EventTableTriggerLogic 9452: layoutX=184, layoutY=128, Operand1=AND 6402, Operand2=AND 6408, Operator=0, Delay=1000
EventTableTriggerLogic 9453: layoutX=184, layoutY=128, Operand1=AND 6402, Operand2=AND 6408, Operator=0, Delay=1000
EventTableTriggerLogic 9454: layoutX=184, layoutY=128, Operand1=AND 6402, Operand2=AND 6408, Operator=0, Delay=1000
EventTableTriggerLogic 9455: layoutX=231, layoutY=144, Operand1=AND 6416, Operand2=pallet1 6426, Operator=0, Delay=1000
EventTableTriggerLogic 9456: layoutX=231, layoutY=144, Operand1=AND 6416, Operand2=pallet1 6426, Operator=0, Delay=1000
EventTableTriggerLogic 9457: layoutX=231, layoutY=144, Operand1=AND 6416, Operand2=pallet1 6426, Operator=0, Delay=1000
EventTableTriggerLogic 9458: layoutX=231, layoutY=144, Operand1=AND 6416, Operand2=pallet1 6426, Operator=0, Delay=1000
EventTableTriggerLogic 9459: layoutX=231, layoutY=144, Operand1=AND 6416, Operand2=pallet1 6426, Operator=0, Delay=1000
EventTableTriggerLogic 9460: layoutX=231, layoutY=144, Operand1=AND 6416, Operand2=pallet1 6426, Operator=0, Delay=1000
EventTableTriggerLogic 9461: layoutX=251, layoutY=143, Operand1=AND 8115, Operand2=pallet3.1 8114, Operator=0, Delay=1000
EventTableTriggerLogic 9462: layoutX=251, layoutY=143, Operand1=AND 8115, Operand2=pallet3.1 8114, Operator=0, Delay=1000
EventTableTriggerLogic 9463: layoutX=251, layoutY=143, Operand1=AND 8115, Operand2=pallet3.1 8114, Operator=0, Delay=1000
EventTableTriggerLogic 9464: layoutX=251, layoutY=143, Operand1=AND 8115, Operand2=pallet3.1 8114, Operator=0, Delay=1000
EventTableTriggerLogic 9465: layoutX=251, layoutY=143, Operand1=AND 8115, Operand2=pallet3.1 8114, Operator=0, Delay=1000
EventTableTriggerLogic 9466: layoutX=251, layoutY=143, Operand1=AND 8115, Operand2=pallet3.1 8114, Operator=0, Delay=1000
EventTableTriggerLogic 9467: layoutX=62, layoutY=38, Operand1=pallet2 8126, Operand2=cellC_slider_horizontal_move 8125, Operator=0, Delay=1000
EventTableTriggerLogic 9468: layoutX=62, layoutY=38, Operand1=pallet2 8126, Operand2=cellC_slider_horizontal_move 8125, Operator=0, Delay=1000
EventTableTriggerLogic 9469: layoutX=62, layoutY=38, Operand1=pallet2 8126, Operand2=cellC_slider_horizontal_move 8125, Operator=0, Delay=1000
EventTableTriggerLogic 9470: layoutX=62, layoutY=38, Operand1=pallet2 8126, Operand2=cellC_slider_horizontal_move 8125, Operator=0, Delay=1000
EventTableTriggerLogic 9471: layoutX=62, layoutY=38, Operand1=pallet2 8126, Operand2=cellC_slider_horizontal_move 8125, Operator=0, Delay=1000
EventTableTriggerLogic 9472: layoutX=62, layoutY=38, Operand1=pallet2 8126, Operand2=cellC_slider_horizontal_move 8125, Operator=0, Delay=1000
EventTableTriggerLogic 9473: layoutX=133, layoutY=37, Operand1=pallet3 6451, Operand2=pose6 6452, Operator=0, Delay=1000
EventTableTriggerLogic 9474: layoutX=133, layoutY=37, Operand1=pallet3 6451, Operand2=pose6 6452, Operator=0, Delay=1000
EventTableTriggerLogic 9475: layoutX=133, layoutY=37, Operand1=pallet3 6451, Operand2=pose6 6452, Operator=0, Delay=1000
EventTableTriggerLogic 9476: layoutX=133, layoutY=37, Operand1=pallet3 6451, Operand2=pose6 6452, Operator=0, Delay=1000
EventTableTriggerLogic 9477: layoutX=133, layoutY=37, Operand1=pallet3 6451, Operand2=pose6 6452, Operator=0, Delay=1000
EventTableTriggerLogic 9478: layoutX=133, layoutY=37, Operand1=pallet3 6451, Operand2=pose6 6452, Operator=0, Delay=1000
EventTableTriggerLogic 9479: layoutX=61, layoutY=50, Operand1=pallet3.2 6456, Operand2=pose3 6457, Operator=0, Delay=1000
EventTableTriggerLogic 9480: layoutX=61, layoutY=50, Operand1=pallet3.2 6456, Operand2=pose3 6457, Operator=0, Delay=1000
EventTableTriggerLogic 9481: layoutX=61, layoutY=50, Operand1=pallet3.2 6456, Operand2=pose3 6457, Operator=0, Delay=1000
EventTableTriggerLogic 9482: layoutX=61, layoutY=50, Operand1=pallet3.2 6456, Operand2=pose3 6457, Operator=0, Delay=1000
EventTableTriggerLogic 9483: layoutX=61, layoutY=50, Operand1=pallet3.2 6456, Operand2=pose3 6457, Operator=0, Delay=1000
EventTableTriggerLogic 9484: layoutX=61, layoutY=50, Operand1=pallet3.2 6456, Operand2=pose3 6457, Operator=0, Delay=1000
EventTableTriggerLogic 9485: layoutX=131, layoutY=52, Operand1=pickpallet1 6461, Operand2=pose7 6462, Operator=0, Delay=1000
EventTableTriggerLogic 9486: layoutX=131, layoutY=52, Operand1=pickpallet1 6461, Operand2=pose7 6462, Operator=0, Delay=1000
EventTableTriggerLogic 9487: layoutX=131, layoutY=52, Operand1=pickpallet1 6461, Operand2=pose7 6462, Operator=0, Delay=1000
EventTableTriggerLogic 9488: layoutX=131, layoutY=52, Operand1=pickpallet1 6461, Operand2=pose7 6462, Operator=0, Delay=1000
EventTableTriggerLogic 9489: layoutX=131, layoutY=52, Operand1=pickpallet1 6461, Operand2=pose7 6462, Operator=0, Delay=1000
EventTableTriggerLogic 9490: layoutX=131, layoutY=52, Operand1=pickpallet1 6461, Operand2=pose7 6462, Operator=0, Delay=1000
EventTableTriggerLogic 9491: layoutX=8, layoutY=16, Operand1=pickpallet2 6466, Operand2=pose13 6467, Operator=0, Delay=1000
EventTableTriggerLogic 9492: layoutX=8, layoutY=16, Operand1=pickpallet2 6466, Operand2=pose13 6467, Operator=0, Delay=1000
EventTableTriggerLogic 9493: layoutX=8, layoutY=16, Operand1=pickpallet2 6466, Operand2=pose13 6467, Operator=0, Delay=1000
EventTableTriggerLogic 9494: layoutX=8, layoutY=16, Operand1=pickpallet2 6466, Operand2=pose13 6467, Operator=0, Delay=1000
EventTableTriggerLogic 9495: layoutX=8, layoutY=16, Operand1=pickpallet2 6466, Operand2=pose13 6467, Operator=0, Delay=1000
EventTableTriggerLogic 9496: layoutX=8, layoutY=16, Operand1=pickpallet2 6466, Operand2=pose13 6467, Operator=0, Delay=1000
EventTableTriggerLogic 9497: layoutX=232, layoutY=117, Operand1=AND 6471, Operand2=pallet4 6481, Operator=0, Delay=1000
EventTableTriggerLogic 9498: layoutX=232, layoutY=117, Operand1=AND 6471, Operand2=pallet4 6481, Operator=0, Delay=1000
EventTableTriggerLogic 9499: layoutX=232, layoutY=117, Operand1=AND 6471, Operand2=pallet4 6481, Operator=0, Delay=1000
EventTableTriggerLogic 9500: layoutX=232, layoutY=117, Operand1=AND 6471, Operand2=pallet4 6481, Operator=0, Delay=1000
EventTableTriggerLogic 9501: layoutX=232, layoutY=117, Operand1=AND 6471, Operand2=pallet4 6481, Operator=0, Delay=1000
EventTableTriggerLogic 9502: layoutX=232, layoutY=117, Operand1=AND 6471, Operand2=pallet4 6481, Operator=0, Delay=1000
EventTableTriggerLogic 9503: layoutX=237, layoutY=122, Operand1=AND 6485, Operand2=conv2_buffer_stopper 6492, Operator=0, Delay=1000
EventTableTriggerLogic 9504: layoutX=237, layoutY=122, Operand1=AND 6485, Operand2=conv2_buffer_stopper 6492, Operator=0, Delay=1000
EventTableTriggerLogic 9505: layoutX=237, layoutY=122, Operand1=AND 6485, Operand2=conv2_buffer_stopper 6492, Operator=0, Delay=1000
EventTableTriggerLogic 9506: layoutX=237, layoutY=122, Operand1=AND 6485, Operand2=conv2_buffer_stopper 6492, Operator=0, Delay=1000
EventTableTriggerLogic 9507: layoutX=237, layoutY=122, Operand1=AND 6485, Operand2=conv2_buffer_stopper 6492, Operator=0, Delay=1000
EventTableTriggerLogic 9508: layoutX=237, layoutY=122, Operand1=AND 6485, Operand2=conv2_buffer_stopper 6492, Operator=0, Delay=1000
EventTableTriggerLogic 9509: layoutX=240, layoutY=90, Operand1=AND 6496, Operand2=AND 6500, Operator=0, Delay=1000
EventTableTriggerLogic 9510: layoutX=240, layoutY=90, Operand1=AND 6496, Operand2=AND 6500, Operator=0, Delay=1000
EventTableTriggerLogic 9511: layoutX=240, layoutY=90, Operand1=AND 6496, Operand2=AND 6500, Operator=0, Delay=1000
EventTableTriggerLogic 9512: layoutX=240, layoutY=90, Operand1=AND 6496, Operand2=AND 6500, Operator=0, Delay=1000
EventTableTriggerLogic 9513: layoutX=240, layoutY=90, Operand1=AND 6496, Operand2=AND 6500, Operator=0, Delay=1000
EventTableTriggerLogic 9514: layoutX=240, layoutY=90, Operand1=AND 6496, Operand2=AND 6500, Operator=0, Delay=1000
EventTableTriggerLogic 9515: layoutX=80, layoutY=49, Operand1=pallet5.1 6513, Operand2=conv2_outer_lifter 6514, Operator=0, Delay=1000
EventTableTriggerLogic 9516: layoutX=80, layoutY=49, Operand1=pallet5.1 6513, Operand2=conv2_outer_lifter 6514, Operator=0, Delay=1000
EventTableTriggerLogic 9517: layoutX=80, layoutY=49, Operand1=pallet5.1 6513, Operand2=conv2_outer_lifter 6514, Operator=0, Delay=1000
EventTableTriggerLogic 9518: layoutX=80, layoutY=49, Operand1=pallet5.1 6513, Operand2=conv2_outer_lifter 6514, Operator=0, Delay=1000
EventTableTriggerLogic 9519: layoutX=80, layoutY=49, Operand1=pallet5.1 6513, Operand2=conv2_outer_lifter 6514, Operator=0, Delay=1000
EventTableTriggerLogic 9520: layoutX=80, layoutY=49, Operand1=pallet5.1 6513, Operand2=conv2_outer_lifter 6514, Operator=0, Delay=1000
EventTableTriggerIO 9521: IOValue=[1], IRC5Controller=? -1, Operator=0, SignalSource=LCFA_profile 1
EventTableTriggerIO 9522: IOValue=[1], IRC5Controller=? -1, Operator=0, SignalSource=LCFA_profile 1
EventTableTriggerIO 9523: IOValue=[1], IRC5Controller=? -1, Operator=0, SignalSource=LCFA_profile 1
EventTableTriggerIO 9524: IOValue=[1], IRC5Controller=? -1, Operator=0, SignalSource=LCFA_profile 1
EventTableTriggerIO 9525: IOValue=[1], IRC5Controller=? -1, Operator=0, SignalSource=LCFA_profile 1
EventTableTriggerIO 9526: IOValue=[1], IRC5Controller=? -1, Operator=0, SignalSource=LCFA_profile 1
EventTableTriggerIO 9527: IOValue=[1], IRC5Controller=? -1, Operator=0, SignalSource=LCFA_profile 1
EventTableTriggerIO 9528: IOValue=[1], IRC5Controller=? -1, Operator=0, SignalSource=LCFA_profile 1
EventTableTriggerIO 9529: IOValue=[1], IRC5Controller=? -1, Operator=0, SignalSource=LCFA_profile 1
EventTableTriggerIO 9530: IOValue=[1], IRC5Controller=? -1, Operator=0, SignalSource=LCFA_profile 1
EventTableTriggerIO 9531: IOValue=[1], IRC5Controller=? -1, Operator=0, SignalSource=LCFA_profile 1
EventTableTriggerIO 9532: IOValue=[1], IRC5Controller=? -1, Operator=0, SignalSource=LCFA_profile 1
EventTableTriggerIO 9533: IOValue=[1], IRC5Controller=? -1, Operator=0, SignalSource=LCFA_profile 1
EventTableTriggerIO 9534: IOValue=[1], IRC5Controller=? -1, Operator=0, SignalSource=LCFA_profile 1
EventTableTriggerIO 9535: IOValue=[1], IRC5Controller=? -1, Operator=0, SignalSource=LCFA_profile 1
EventTableTriggerIO 9536: IOValue=[1], IRC5Controller=? -1, Operator=0, SignalSource=LCFA_profile 1
EventTableTriggerIO 9537: IOValue=[1], IRC5Controller=? -1, Operator=0, SignalSource=LCFA_profile 1
EventTableTriggerIO 9538: IOValue=[1], IRC5Controller=? -1, Operator=0, SignalSource=LCFA_profile 1
EventTableTriggerIO 9539: IOValue=[1], IRC5Controller=? -1, Operator=0, SignalSource=LCFA_profile 1
EventTableTriggerIO 9540: IOValue=[1], IRC5Controller=? -1, Operator=0, SignalSource=LCFA_profile 1
EventTableTriggerIO 9541: IOValue=[1], IRC5Controller=? -1, Operator=0, SignalSource=LCFA_profile 1
EventTableTriggerIO 9542: IOValue=[1], IRC5Controller=? -1, Operator=0, SignalSource=LCFA_profile 1
EventTableTriggerIO 9543: IOValue=[1], IRC5Controller=? -1, Operator=0, SignalSource=LCFA_profile 1
EventTableTriggerIO 9544: IOValue=[1], IRC5Controller=? -1, Operator=0, SignalSource=LCFA_profile 1
EventTableTriggerIO 9545: IOValue=[1], IRC5Controller=? -1, Operator=0, SignalSource=LCFA_profile 1
EventTableTriggerIO 9546: IOValue=[1], IRC5Controller=? -1, Operator=0, SignalSource=LCFA_profile 1
EventTableTriggerIO 9547: IOValue=[1], IRC5Controller=? -1, Operator=0, SignalSource=LCFA_profile 1
EventTableTriggerIO 9548: IOValue=[1], IRC5Controller=? -1, Operator=0, SignalSource=LCFA_profile 1
EventTableTriggerIO 9549: IOValue=[1], IRC5Controller=? -1, Operator=0, SignalSource=LCFA_profile 1
EventTableTriggerIO 9550: IOValue=[1], IRC5Controller=? -1, Operator=0, SignalSource=LCFA_profile 1
EventTableTriggerIO 9551: IOValue=[1], IRC5Controller=? -1, Operator=0, SignalSource=LCFA_profile 1
EventTableTriggerIO 9552: IOValue=[1], IRC5Controller=? -1, Operator=0, SignalSource=LCFA_profile 1
EventTableTriggerIO 9553: IOValue=[1], IRC5Controller=? -1, Operator=0, SignalSource=LCFA_profile 1
EventTableTriggerIO 9554: IOValue=[1], IRC5Controller=? -1, Operator=0, SignalSource=LCFA_profile 1
EventTableTriggerIO 9555: IOValue=[1], IRC5Controller=? -1, Operator=0, SignalSource=LCFA_profile 1
EventTableTriggerIO 9556: IOValue=[1], IRC5Controller=? -1, Operator=0, SignalSource=LCFA_profile 1
EventTableTriggerIO 9557: IOValue=[1], IRC5Controller=? -1, Operator=0, SignalSource=LCFA_profile 1
EventTableTriggerIO 9558: IOValue=[1], IRC5Controller=? -1, Operator=0, SignalSource=LCFA_profile 1
EventTableTriggerIO 9559: IOValue=[1], IRC5Controller=? -1, Operator=0, SignalSource=LCFA_profile 1
EventTableTriggerIO 9560: IOValue=[1], IRC5Controller=? -1, Operator=0, SignalSource=LCFA_profile 1
EventTableTriggerIO 9561: IOValue=[1], IRC5Controller=? -1, Operator=0, SignalSource=LCFA_profile 1
EventTableTriggerIO 9562: IOValue=[1], IRC5Controller=? -1, Operator=0, SignalSource=LCFA_profile 1
EventTableTriggerIO 9563: IOValue=[1], IRC5Controller=? -1, Operator=0, SignalSource=LCFA_profile 1
EventTableTriggerIO 9564: IOValue=[1], IRC5Controller=? -1, Operator=0, SignalSource=LCFA_profile 1
EventTableTriggerIO 9565: IOValue=[1], IRC5Controller=? -1, Operator=0, SignalSource=LCFA_profile 1
EventTableTriggerIO 9566: IOValue=[1], IRC5Controller=? -1, Operator=0, SignalSource=LCFA_profile 1
EventTableTriggerIO 9567: IOValue=[1], IRC5Controller=? -1, Operator=0, SignalSource=LCFA_profile 1
EventTableTriggerIO 9568: IOValue=[1], IRC5Controller=? -1, Operator=0, SignalSource=LCFA_profile 1
EventTableTriggerIO 9569: IOValue=[1], IRC5Controller=? -1, Operator=0, SignalSource=LCFA_profile 1
EventTableTriggerIO 9570: IOValue=[1], IRC5Controller=? -1, Operator=0, SignalSource=LCFA_profile 1
EventTableTriggerIO 9571: IOValue=[1], IRC5Controller=? -1, Operator=0, SignalSource=LCFA_profile 1
EventTableTriggerIO 9572: IOValue=[1], IRC5Controller=? -1, Operator=0, SignalSource=LCFA_profile 1
EventTableTriggerIO 9573: IOValue=[1], IRC5Controller=? -1, Operator=0, SignalSource=LCFA_profile 1
EventTableTriggerIO 9574: IOValue=[1], IRC5Controller=? -1, Operator=0, SignalSource=LCFA_profile 1
EventTableTriggerIO 9575: IOValue=[1], IRC5Controller=? -1, Operator=0, SignalSource=LCFA_profile 1
EventTableTriggerIO 9576: IOValue=[1], IRC5Controller=? -1, Operator=0, SignalSource=LCFA_profile 1
EventTableTriggerIO 9577: IOValue=[1], IRC5Controller=? -1, Operator=0, SignalSource=LCFA_profile 1
EventTableTriggerIO 9578: IOValue=[1], IRC5Controller=? -1, Operator=0, SignalSource=LCFA_profile 1
EventTableTriggerIO 9579: IOValue=[1], IRC5Controller=? -1, Operator=0, SignalSource=LCFA_profile 1
EventTableTriggerIO 9580: IOValue=[1], IRC5Controller=? -1, Operator=0, SignalSource=LCFA_profile 1
EventTableTriggerIO 9581: IOValue=[0], IRC5Controller=? -1, Operator=0, SignalSource=ALab_CellC_v1.0_4 5362
EventTableTriggerIO 9582: IOValue=[0], IRC5Controller=? -1, Operator=0, SignalSource=ALab_CellC_v1.0_4 5362
EventTableTriggerIO 9583: IOValue=[0], IRC5Controller=? -1, Operator=0, SignalSource=ALab_CellC_v1.0_4 5362
EventTableTriggerIO 9584: IOValue=[0], IRC5Controller=? -1, Operator=0, SignalSource=ALab_CellC_v1.0_4 5362
EventTableTriggerIO 9585: IOValue=[0], IRC5Controller=? -1, Operator=0, SignalSource=ALab_CellC_v1.0_4 5362
EventTableTriggerIO 9586: IOValue=[0], IRC5Controller=? -1, Operator=0, SignalSource=ALab_CellC_v1.0_4 5362
EventTableTriggerIO 9587: IOValue=[1], IRC5Controller=? -1, Operator=0, SignalSource=ALab_CellC_v1.0_4 5362
EventTableTriggerIO 9588: IOValue=[1], IRC5Controller=? -1, Operator=0, SignalSource=ALab_CellC_v1.0_4 5362
EventTableTriggerIO 9589: IOValue=[1], IRC5Controller=? -1, Operator=0, SignalSource=ALab_CellC_v1.0_4 5362
EventTableTriggerIO 9590: IOValue=[1], IRC5Controller=? -1, Operator=0, SignalSource=ALab_CellC_v1.0_4 5362
EventTableTriggerIO 9591: IOValue=[1], IRC5Controller=? -1, Operator=0, SignalSource=ALab_CellC_v1.0_4 5362
EventTableTriggerIO 9592: IOValue=[1], IRC5Controller=? -1, Operator=0, SignalSource=ALab_CellC_v1.0_4 5362
EventTableTriggerIO 9593: IOValue=[0], IRC5Controller=? -1, Operator=0, SignalSource=ALab_CellC_v1.0_4 5362
EventTableTriggerIO 9594: IOValue=[0], IRC5Controller=? -1, Operator=0, SignalSource=ALab_CellC_v1.0_4 5362
EventTableTriggerIO 9595: IOValue=[0], IRC5Controller=? -1, Operator=0, SignalSource=ALab_CellC_v1.0_4 5362
EventTableTriggerIO 9596: IOValue=[0], IRC5Controller=? -1, Operator=0, SignalSource=ALab_CellC_v1.0_4 5362
EventTableTriggerIO 9597: IOValue=[0], IRC5Controller=? -1, Operator=0, SignalSource=ALab_CellC_v1.0_4 5362
EventTableTriggerIO 9598: IOValue=[0], IRC5Controller=? -1, Operator=0, SignalSource=ALab_CellC_v1.0_4 5362
EventTableTriggerIO 9599: IOValue=[1], IRC5Controller=? -1, Operator=0, SignalSource=ALab_CellC_v1.0_4 5362
EventTableTriggerIO 9600: IOValue=[1], IRC5Controller=? -1, Operator=0, SignalSource=ALab_CellC_v1.0_4 5362
EventTableTriggerIO 9601: IOValue=[1], IRC5Controller=? -1, Operator=0, SignalSource=ALab_CellC_v1.0_4 5362
EventTableTriggerIO 9602: IOValue=[1], IRC5Controller=? -1, Operator=0, SignalSource=ALab_CellC_v1.0_4 5362
EventTableTriggerIO 9603: IOValue=[1], IRC5Controller=? -1, Operator=0, SignalSource=ALab_CellC_v1.0_4 5362
EventTableTriggerIO 9604: IOValue=[1], IRC5Controller=? -1, Operator=0, SignalSource=ALab_CellC_v1.0_4 5362
EventTableTriggerIO 9605: IOValue=[1], IRC5Controller=? -1, Operator=0, SignalSource=ALab_CellC_v1.0_4 5362
EventTableTriggerIO 9606: IOValue=[1], IRC5Controller=? -1, Operator=0, SignalSource=ALab_CellC_v1.0_4 5362
EventTableTriggerIO 9607: IOValue=[1], IRC5Controller=? -1, Operator=0, SignalSource=ALab_CellC_v1.0_4 5362
EventTableTriggerIO 9608: IOValue=[1], IRC5Controller=? -1, Operator=0, SignalSource=ALab_CellC_v1.0_4 5362
EventTableTriggerIO 9609: IOValue=[1], IRC5Controller=? -1, Operator=0, SignalSource=ALab_CellC_v1.0_4 5362
EventTableTriggerIO 9610: IOValue=[1], IRC5Controller=? -1, Operator=0, SignalSource=ALab_CellC_v1.0_4 5362
EventTableTriggerIO 9611: IOValue=[0], IRC5Controller=? -1, Operator=0, SignalSource=ALab_CellC_v1.0_4 5362
EventTableTriggerIO 9612: IOValue=[0], IRC5Controller=? -1, Operator=0, SignalSource=ALab_CellC_v1.0_4 5362
EventTableTriggerIO 9613: IOValue=[0], IRC5Controller=? -1, Operator=0, SignalSource=ALab_CellC_v1.0_4 5362
EventTableTriggerIO 9614: IOValue=[0], IRC5Controller=? -1, Operator=0, SignalSource=ALab_CellC_v1.0_4 5362
EventTableTriggerIO 9615: IOValue=[0], IRC5Controller=? -1, Operator=0, SignalSource=ALab_CellC_v1.0_4 5362
EventTableTriggerIO 9616: IOValue=[0], IRC5Controller=? -1, Operator=0, SignalSource=ALab_CellC_v1.0_4 5362
EventTableTriggerIO 9617: IOValue=[0], IRC5Controller=? -1, Operator=0, SignalSource=ALab_CellC_v1.0_4 5362
EventTableTriggerIO 9618: IOValue=[0], IRC5Controller=? -1, Operator=0, SignalSource=ALab_CellC_v1.0_4 5362
EventTableTriggerIO 9619: IOValue=[0], IRC5Controller=? -1, Operator=0, SignalSource=ALab_CellC_v1.0_4 5362
EventTableTriggerIO 9620: IOValue=[0], IRC5Controller=? -1, Operator=0, SignalSource=ALab_CellC_v1.0_4 5362
EventTableTriggerIO 9621: IOValue=[0], IRC5Controller=? -1, Operator=0, SignalSource=ALab_CellC_v1.0_4 5362
EventTableTriggerIO 9622: IOValue=[0], IRC5Controller=? -1, Operator=0, SignalSource=ALab_CellC_v1.0_4 5362
EventTableTriggerIO 9623: IOValue=[1], IRC5Controller=? -1, Operator=0, SignalSource=ALab_CellC_v1.0_4 5362
EventTableTriggerIO 9624: IOValue=[1], IRC5Controller=? -1, Operator=0, SignalSource=ALab_CellC_v1.0_4 5362
EventTableTriggerIO 9625: IOValue=[1], IRC5Controller=? -1, Operator=0, SignalSource=ALab_CellC_v1.0_4 5362
EventTableTriggerIO 9626: IOValue=[1], IRC5Controller=? -1, Operator=0, SignalSource=ALab_CellC_v1.0_4 5362
EventTableTriggerIO 9627: IOValue=[1], IRC5Controller=? -1, Operator=0, SignalSource=ALab_CellC_v1.0_4 5362
EventTableTriggerIO 9628: IOValue=[1], IRC5Controller=? -1, Operator=0, SignalSource=ALab_CellC_v1.0_4 5362
EventTableTriggerIO 9629: IOValue=[1], IRC5Controller=? -1, Operator=0, SignalSource=ALab_CellC_v1.0_4 5362
EventTableTriggerIO 9630: IOValue=[1], IRC5Controller=? -1, Operator=0, SignalSource=ALab_CellC_v1.0_4 5362
EventTableTriggerIO 9631: IOValue=[1], IRC5Controller=? -1, Operator=0, SignalSource=ALab_CellC_v1.0_4 5362
EventTableTriggerIO 9632: IOValue=[1], IRC5Controller=? -1, Operator=0, SignalSource=ALab_CellC_v1.0_4 5362
EventTableTriggerIO 9633: IOValue=[1], IRC5Controller=? -1, Operator=0, SignalSource=ALab_CellC_v1.0_4 5362
EventTableTriggerIO 9634: IOValue=[1], IRC5Controller=? -1, Operator=0, SignalSource=ALab_CellC_v1.0_4 5362
EventTableTriggerIO 9635: IOValue=[0], IRC5Controller=? -1, Operator=0, SignalSource=ALab_CellC_v1.0_4 5362
EventTableTriggerIO 9636: IOValue=[0], IRC5Controller=? -1, Operator=0, SignalSource=ALab_CellC_v1.0_4 5362
EventTableTriggerIO 9637: IOValue=[0], IRC5Controller=? -1, Operator=0, SignalSource=ALab_CellC_v1.0_4 5362
EventTableTriggerIO 9638: IOValue=[0], IRC5Controller=? -1, Operator=0, SignalSource=ALab_CellC_v1.0_4 5362
EventTableTriggerIO 9639: IOValue=[0], IRC5Controller=? -1, Operator=0, SignalSource=ALab_CellC_v1.0_4 5362
EventTableTriggerIO 9640: IOValue=[0], IRC5Controller=? -1, Operator=0, SignalSource=ALab_CellC_v1.0_4 5362
EventTableTriggerIO 9641: IOValue=[1], IRC5Controller=? -1, Operator=0, SignalSource=ALab_CellC_v1.0_4 5362
EventTableTriggerIO 9642: IOValue=[1], IRC5Controller=? -1, Operator=0, SignalSource=ALab_CellC_v1.0_4 5362
EventTableTriggerIO 9643: IOValue=[1], IRC5Controller=? -1, Operator=0, SignalSource=ALab_CellC_v1.0_4 5362
EventTableTriggerIO 9644: IOValue=[1], IRC5Controller=? -1, Operator=0, SignalSource=ALab_CellC_v1.0_4 5362
EventTableTriggerIO 9645: IOValue=[1], IRC5Controller=? -1, Operator=0, SignalSource=ALab_CellC_v1.0_4 5362
EventTableTriggerIO 9646: IOValue=[1], IRC5Controller=? -1, Operator=0, SignalSource=ALab_CellC_v1.0_4 5362
EventTableTriggerIO 9647: IOValue=[0], IRC5Controller=? -1, Operator=0, SignalSource=ALab_CellC_v1.0_4 5362
EventTableTriggerIO 9648: IOValue=[0], IRC5Controller=? -1, Operator=0, SignalSource=ALab_CellC_v1.0_4 5362
EventTableTriggerIO 9649: IOValue=[0], IRC5Controller=? -1, Operator=0, SignalSource=ALab_CellC_v1.0_4 5362
EventTableTriggerIO 9650: IOValue=[0], IRC5Controller=? -1, Operator=0, SignalSource=ALab_CellC_v1.0_4 5362
EventTableTriggerIO 9651: IOValue=[0], IRC5Controller=? -1, Operator=0, SignalSource=ALab_CellC_v1.0_4 5362
EventTableTriggerIO 9652: IOValue=[0], IRC5Controller=? -1, Operator=0, SignalSource=ALab_CellC_v1.0_4 5362
EventTableTriggerIO 9653: IOValue=[0], IRC5Controller=? -1, Operator=0, SignalSource=ALab_CellC_v1.0_4 5362
EventTableTriggerIO 9654: IOValue=[0], IRC5Controller=? -1, Operator=0, SignalSource=ALab_CellC_v1.0_4 5362
EventTableTriggerIO 9655: IOValue=[0], IRC5Controller=? -1, Operator=0, SignalSource=ALab_CellC_v1.0_4 5362
EventTableTriggerIO 9656: IOValue=[0], IRC5Controller=? -1, Operator=0, SignalSource=ALab_CellC_v1.0_4 5362
EventTableTriggerIO 9657: IOValue=[0], IRC5Controller=? -1, Operator=0, SignalSource=ALab_CellC_v1.0_4 5362
EventTableTriggerIO 9658: IOValue=[0], IRC5Controller=? -1, Operator=0, SignalSource=ALab_CellC_v1.0_4 5362
EventTableTriggerIO 9659: IOValue=[1], IRC5Controller=? -1, Operator=0, SignalSource=ALab_CellC_v1.0_4 5362
EventTableTriggerIO 9660: IOValue=[1], IRC5Controller=? -1, Operator=0, SignalSource=ALab_CellC_v1.0_4 5362
EventTableTriggerIO 9661: IOValue=[1], IRC5Controller=? -1, Operator=0, SignalSource=ALab_CellC_v1.0_4 5362
EventTableTriggerIO 9662: IOValue=[1], IRC5Controller=? -1, Operator=0, SignalSource=ALab_CellC_v1.0_4 5362
EventTableTriggerIO 9663: IOValue=[1], IRC5Controller=? -1, Operator=0, SignalSource=ALab_CellC_v1.0_4 5362
EventTableTriggerIO 9664: IOValue=[1], IRC5Controller=? -1, Operator=0, SignalSource=ALab_CellC_v1.0_4 5362
EventTableTriggerIO 9665: IOValue=[1], IRC5Controller=? -1, Operator=0, SignalSource=ALab_CellC_v1.0_4 5362
EventTableTriggerIO 9666: IOValue=[1], IRC5Controller=? -1, Operator=0, SignalSource=ALab_CellC_v1.0_4 5362
EventTableTriggerIO 9667: IOValue=[1], IRC5Controller=? -1, Operator=0, SignalSource=ALab_CellC_v1.0_4 5362
EventTableTriggerIO 9668: IOValue=[1], IRC5Controller=? -1, Operator=0, SignalSource=ALab_CellC_v1.0_4 5362
EventTableTriggerIO 9669: IOValue=[1], IRC5Controller=? -1, Operator=0, SignalSource=ALab_CellC_v1.0_4 5362
EventTableTriggerIO 9670: IOValue=[1], IRC5Controller=? -1, Operator=0, SignalSource=ALab_CellC_v1.0_4 5362
EventTableTriggerIO 9671: IOValue=[0], IRC5Controller=? -1, Operator=0, SignalSource=ALab_CellC_v1.0_4 5362
EventTableTriggerIO 9672: IOValue=[0], IRC5Controller=? -1, Operator=0, SignalSource=ALab_CellC_v1.0_4 5362
EventTableTriggerIO 9673: IOValue=[0], IRC5Controller=? -1, Operator=0, SignalSource=ALab_CellC_v1.0_4 5362
EventTableTriggerIO 9674: IOValue=[0], IRC5Controller=? -1, Operator=0, SignalSource=ALab_CellC_v1.0_4 5362
EventTableTriggerIO 9675: IOValue=[0], IRC5Controller=? -1, Operator=0, SignalSource=ALab_CellC_v1.0_4 5362
EventTableTriggerIO 9676: IOValue=[0], IRC5Controller=? -1, Operator=0, SignalSource=ALab_CellC_v1.0_4 5362
EventTableTriggerIO 9677: IOValue=[0], IRC5Controller=? -1, Operator=0, SignalSource=ALab_CellC_v1.0_4 5362
EventTableTriggerIO 9678: IOValue=[0], IRC5Controller=? -1, Operator=0, SignalSource=ALab_CellC_v1.0_4 5362
EventTableTriggerIO 9679: IOValue=[0], IRC5Controller=? -1, Operator=0, SignalSource=ALab_CellC_v1.0_4 5362
EventTableTriggerIO 9680: IOValue=[0], IRC5Controller=? -1, Operator=0, SignalSource=ALab_CellC_v1.0_4 5362
EventTableTriggerIO 9681: IOValue=[0], IRC5Controller=? -1, Operator=0, SignalSource=ALab_CellC_v1.0_4 5362
EventTableTriggerIO 9682: IOValue=[0], IRC5Controller=? -1, Operator=0, SignalSource=ALab_CellC_v1.0_4 5362
EventTableTriggerIO 9683: IOValue=[1], IRC5Controller=? -1, Operator=0, SignalSource=ALab_CellC_v1.0_4 5362
EventTableTriggerIO 9684: IOValue=[1], IRC5Controller=? -1, Operator=0, SignalSource=ALab_CellC_v1.0_4 5362
EventTableTriggerIO 9685: IOValue=[1], IRC5Controller=? -1, Operator=0, SignalSource=ALab_CellC_v1.0_4 5362
EventTableTriggerIO 9686: IOValue=[1], IRC5Controller=? -1, Operator=0, SignalSource=ALab_CellC_v1.0_4 5362
EventTableTriggerIO 9687: IOValue=[1], IRC5Controller=? -1, Operator=0, SignalSource=ALab_CellC_v1.0_4 5362
EventTableTriggerIO 9688: IOValue=[1], IRC5Controller=? -1, Operator=0, SignalSource=ALab_CellC_v1.0_4 5362
EventTableTriggerIO 9689: IOValue=[1], IRC5Controller=? -1, Operator=0, SignalSource=ALab_CellC_v1.0_4 5362
EventTableTriggerIO 9690: IOValue=[1], IRC5Controller=? -1, Operator=0, SignalSource=ALab_CellC_v1.0_4 5362
EventTableTriggerIO 9691: IOValue=[1], IRC5Controller=? -1, Operator=0, SignalSource=ALab_CellC_v1.0_4 5362
EventTableTriggerIO 9692: IOValue=[1], IRC5Controller=? -1, Operator=0, SignalSource=ALab_CellC_v1.0_4 5362
EventTableTriggerIO 9693: IOValue=[1], IRC5Controller=? -1, Operator=0, SignalSource=ALab_CellC_v1.0_4 5362
EventTableTriggerIO 9694: IOValue=[1], IRC5Controller=? -1, Operator=0, SignalSource=ALab_CellC_v1.0_4 5362
EventTableTriggerIO 9695: IOValue=[0], IRC5Controller=? -1, Operator=0, SignalSource=ALab_CellC_v1.0_4 5362
EventTableTriggerIO 9696: IOValue=[0], IRC5Controller=? -1, Operator=0, SignalSource=ALab_CellC_v1.0_4 5362
EventTableTriggerIO 9697: IOValue=[0], IRC5Controller=? -1, Operator=0, SignalSource=ALab_CellC_v1.0_4 5362
EventTableTriggerIO 9698: IOValue=[0], IRC5Controller=? -1, Operator=0, SignalSource=ALab_CellC_v1.0_4 5362
EventTableTriggerIO 9699: IOValue=[0], IRC5Controller=? -1, Operator=0, SignalSource=ALab_CellC_v1.0_4 5362
EventTableTriggerIO 9700: IOValue=[0], IRC5Controller=? -1, Operator=0, SignalSource=ALab_CellC_v1.0_4 5362
EventTableTriggerIO 9701: IOValue=[1], IRC5Controller=? -1, Operator=0, SignalSource=LCFA_profile 1
EventTableTriggerIO 9702: IOValue=[1], IRC5Controller=? -1, Operator=0, SignalSource=LCFA_profile 1
EventTableTriggerIO 9703: IOValue=[1], IRC5Controller=? -1, Operator=0, SignalSource=LCFA_profile 1
EventTableTriggerIO 9704: IOValue=[1], IRC5Controller=? -1, Operator=0, SignalSource=LCFA_profile 1
EventTableTriggerIO 9705: IOValue=[1], IRC5Controller=? -1, Operator=0, SignalSource=LCFA_profile 1
EventTableTriggerIO 9706: IOValue=[1], IRC5Controller=? -1, Operator=0, SignalSource=LCFA_profile 1
EventTableTriggerIO 9707: IOValue=[1], IRC5Controller=? -1, Operator=0, SignalSource=LCFA_profile 1
EventTableTriggerIO 9708: IOValue=[1], IRC5Controller=? -1, Operator=0, SignalSource=LCFA_profile 1
EventTableTriggerIO 9709: IOValue=[1], IRC5Controller=? -1, Operator=0, SignalSource=LCFA_profile 1
EventTableTriggerIO 9710: IOValue=[1], IRC5Controller=? -1, Operator=0, SignalSource=LCFA_profile 1
EventTableTriggerIO 9711: IOValue=[1], IRC5Controller=? -1, Operator=0, SignalSource=LCFA_profile 1
EventTableTriggerIO 9712: IOValue=[1], IRC5Controller=? -1, Operator=0, SignalSource=LCFA_profile 1
EventTableTriggerIO 9713: IOValue=[1], IRC5Controller=? -1, Operator=0, SignalSource=LCFA_profile 1
EventTableTriggerIO 9714: IOValue=[1], IRC5Controller=? -1, Operator=0, SignalSource=LCFA_profile 1
EventTableTriggerIO 9715: IOValue=[1], IRC5Controller=? -1, Operator=0, SignalSource=LCFA_profile 1
EventTableTriggerIO 9716: IOValue=[1], IRC5Controller=? -1, Operator=0, SignalSource=LCFA_profile 1
EventTableTriggerIO 9717: IOValue=[1], IRC5Controller=? -1, Operator=0, SignalSource=LCFA_profile 1
EventTableTriggerIO 9718: IOValue=[1], IRC5Controller=? -1, Operator=0, SignalSource=LCFA_profile 1
EventTableTriggerIO 9719: IOValue=[1], IRC5Controller=? -1, Operator=0, SignalSource=LCFA_profile 1
EventTableTriggerIO 9720: IOValue=[1], IRC5Controller=? -1, Operator=0, SignalSource=LCFA_profile 1
EventTableTriggerIO 9721: IOValue=[1], IRC5Controller=? -1, Operator=0, SignalSource=LCFA_profile 1
EventTableTriggerIO 9722: IOValue=[1], IRC5Controller=? -1, Operator=0, SignalSource=LCFA_profile 1
EventTableTriggerIO 9723: IOValue=[1], IRC5Controller=? -1, Operator=0, SignalSource=LCFA_profile 1
EventTableTriggerIO 9724: IOValue=[1], IRC5Controller=? -1, Operator=0, SignalSource=LCFA_profile 1
EventTableTriggerIO 9725: IOValue=[1], IRC5Controller=? -1, Operator=0, SignalSource=ALab_CellC_v1.0_4 5362
EventTableTriggerIO 9726: IOValue=[1], IRC5Controller=? -1, Operator=0, SignalSource=ALab_CellC_v1.0_4 5362
EventTableTriggerIO 9727: IOValue=[1], IRC5Controller=? -1, Operator=0, SignalSource=ALab_CellC_v1.0_4 5362
EventTableTriggerIO 9728: IOValue=[1], IRC5Controller=? -1, Operator=0, SignalSource=ALab_CellC_v1.0_4 5362
EventTableTriggerIO 9729: IOValue=[1], IRC5Controller=? -1, Operator=0, SignalSource=ALab_CellC_v1.0_4 5362
EventTableTriggerIO 9730: IOValue=[1], IRC5Controller=? -1, Operator=0, SignalSource=ALab_CellC_v1.0_4 5362
EventTableTriggerIO 9731: IOValue=[0], IRC5Controller=? -1, Operator=0, SignalSource=ALab_CellC_v1.0_4 5362
EventTableTriggerIO 9732: IOValue=[0], IRC5Controller=? -1, Operator=0, SignalSource=ALab_CellC_v1.0_4 5362
EventTableTriggerIO 9733: IOValue=[0], IRC5Controller=? -1, Operator=0, SignalSource=ALab_CellC_v1.0_4 5362
EventTableTriggerIO 9734: IOValue=[0], IRC5Controller=? -1, Operator=0, SignalSource=ALab_CellC_v1.0_4 5362
EventTableTriggerIO 9735: IOValue=[0], IRC5Controller=? -1, Operator=0, SignalSource=ALab_CellC_v1.0_4 5362
EventTableTriggerIO 9736: IOValue=[0], IRC5Controller=? -1, Operator=0, SignalSource=ALab_CellC_v1.0_4 5362
EventTableTriggerIO 9737: IOValue=[1], IRC5Controller=? -1, Operator=0, SignalSource=LCFA_profile 1
EventTableTriggerIO 9738: IOValue=[1], IRC5Controller=? -1, Operator=0, SignalSource=LCFA_profile 1
EventTableTriggerIO 9739: IOValue=[1], IRC5Controller=? -1, Operator=0, SignalSource=LCFA_profile 1
EventTableTriggerIO 9740: IOValue=[1], IRC5Controller=? -1, Operator=0, SignalSource=LCFA_profile 1
EventTableTriggerIO 9741: IOValue=[1], IRC5Controller=? -1, Operator=0, SignalSource=LCFA_profile 1
EventTableTriggerIO 9742: IOValue=[1], IRC5Controller=? -1, Operator=0, SignalSource=LCFA_profile 1
EventTableTriggerIO 9743: IOValue=[1], IRC5Controller=? -1, Operator=0, SignalSource=LCFA_profile 1
EventTableTriggerIO 9744: IOValue=[1], IRC5Controller=? -1, Operator=0, SignalSource=LCFA_profile 1
EventTableTriggerIO 9745: IOValue=[1], IRC5Controller=? -1, Operator=0, SignalSource=LCFA_profile 1
EventTableTriggerIO 9746: IOValue=[1], IRC5Controller=? -1, Operator=0, SignalSource=LCFA_profile 1
EventTableTriggerIO 9747: IOValue=[1], IRC5Controller=? -1, Operator=0, SignalSource=LCFA_profile 1
EventTableTriggerIO 9748: IOValue=[1], IRC5Controller=? -1, Operator=0, SignalSource=LCFA_profile 1
EventTableTriggerIO 9749: IOValue=[1], IRC5Controller=? -1, Operator=0, SignalSource=LCFA_profile 1
EventTableTriggerIO 9750: IOValue=[1], IRC5Controller=? -1, Operator=0, SignalSource=LCFA_profile 1
EventTableTriggerIO 9751: IOValue=[1], IRC5Controller=? -1, Operator=0, SignalSource=LCFA_profile 1
EventTableTriggerIO 9752: IOValue=[1], IRC5Controller=? -1, Operator=0, SignalSource=LCFA_profile 1
EventTableTriggerIO 9753: IOValue=[1], IRC5Controller=? -1, Operator=0, SignalSource=LCFA_profile 1
EventTableTriggerIO 9754: IOValue=[1], IRC5Controller=? -1, Operator=0, SignalSource=LCFA_profile 1
EventTableTriggerIO 9755: IOValue=[1], IRC5Controller=? -1, Operator=0, SignalSource=LCFA_profile 1
EventTableTriggerIO 9756: IOValue=[1], IRC5Controller=? -1, Operator=0, SignalSource=LCFA_profile 1
EventTableTriggerIO 9757: IOValue=[1], IRC5Controller=? -1, Operator=0, SignalSource=LCFA_profile 1
EventTableTriggerIO 9758: IOValue=[1], IRC5Controller=? -1, Operator=0, SignalSource=LCFA_profile 1
EventTableTriggerIO 9759: IOValue=[1], IRC5Controller=? -1, Operator=0, SignalSource=LCFA_profile 1
EventTableTriggerIO 9760: IOValue=[1], IRC5Controller=? -1, Operator=0, SignalSource=LCFA_profile 1
EventTableTriggerIO 9761: IOValue=[1], IRC5Controller=? -1, Operator=0, SignalSource=ALab_CellC_v1.0_4 5362
EventTableTriggerIO 9762: IOValue=[1], IRC5Controller=? -1, Operator=0, SignalSource=ALab_CellC_v1.0_4 5362
EventTableTriggerIO 9763: IOValue=[1], IRC5Controller=? -1, Operator=0, SignalSource=ALab_CellC_v1.0_4 5362
EventTableTriggerIO 9764: IOValue=[1], IRC5Controller=? -1, Operator=0, SignalSource=ALab_CellC_v1.0_4 5362
EventTableTriggerIO 9765: IOValue=[1], IRC5Controller=? -1, Operator=0, SignalSource=ALab_CellC_v1.0_4 5362
EventTableTriggerIO 9766: IOValue=[1], IRC5Controller=? -1, Operator=0, SignalSource=ALab_CellC_v1.0_4 5362
EventTableTriggerIO 9767: IOValue=[0], IRC5Controller=? -1, Operator=0, SignalSource=ALab_CellC_v1.0_4 5362
EventTableTriggerIO 9768: IOValue=[0], IRC5Controller=? -1, Operator=0, SignalSource=ALab_CellC_v1.0_4 5362
EventTableTriggerIO 9769: IOValue=[0], IRC5Controller=? -1, Operator=0, SignalSource=ALab_CellC_v1.0_4 5362
EventTableTriggerIO 9770: IOValue=[0], IRC5Controller=? -1, Operator=0, SignalSource=ALab_CellC_v1.0_4 5362
EventTableTriggerIO 9771: IOValue=[0], IRC5Controller=? -1, Operator=0, SignalSource=ALab_CellC_v1.0_4 5362
EventTableTriggerIO 9772: IOValue=[0], IRC5Controller=? -1, Operator=0, SignalSource=ALab_CellC_v1.0_4 5362
EventTableTriggerIO 9773: IOValue=[1], IRC5Controller=? -1, Operator=0, SignalSource=ALab_CellC_v1.0_4 5362
EventTableTriggerIO 9774: IOValue=[1], IRC5Controller=? -1, Operator=0, SignalSource=ALab_CellC_v1.0_4 5362
EventTableTriggerIO 9775: IOValue=[1], IRC5Controller=? -1, Operator=0, SignalSource=ALab_CellC_v1.0_4 5362
EventTableTriggerIO 9776: IOValue=[1], IRC5Controller=? -1, Operator=0, SignalSource=ALab_CellC_v1.0_4 5362
EventTableTriggerIO 9777: IOValue=[1], IRC5Controller=? -1, Operator=0, SignalSource=ALab_CellC_v1.0_4 5362
EventTableTriggerIO 9778: IOValue=[1], IRC5Controller=? -1, Operator=0, SignalSource=ALab_CellC_v1.0_4 5362
EventTableTriggerIO 9779: IOValue=[0], IRC5Controller=? -1, Operator=0, SignalSource=ALab_CellC_v1.0_4 5362
EventTableTriggerIO 9780: IOValue=[0], IRC5Controller=? -1, Operator=0, SignalSource=ALab_CellC_v1.0_4 5362
EventTableTriggerIO 9781: IOValue=[0], IRC5Controller=? -1, Operator=0, SignalSource=ALab_CellC_v1.0_4 5362
EventTableTriggerIO 9782: IOValue=[0], IRC5Controller=? -1, Operator=0, SignalSource=ALab_CellC_v1.0_4 5362
EventTableTriggerIO 9783: IOValue=[0], IRC5Controller=? -1, Operator=0, SignalSource=ALab_CellC_v1.0_4 5362
EventTableTriggerIO 9784: IOValue=[0], IRC5Controller=? -1, Operator=0, SignalSource=ALab_CellC_v1.0_4 5362
EventTableTriggerIO 9785: IOValue=[0], IRC5Controller=? -1, Operator=0, SignalSource=ALab_CellC_v1.0_4 5362
EventTableTriggerIO 9786: IOValue=[0], IRC5Controller=? -1, Operator=0, SignalSource=ALab_CellC_v1.0_4 5362
EventTableTriggerIO 9787: IOValue=[0], IRC5Controller=? -1, Operator=0, SignalSource=ALab_CellC_v1.0_4 5362
EventTableTriggerIO 9788: IOValue=[0], IRC5Controller=? -1, Operator=0, SignalSource=ALab_CellC_v1.0_4 5362
EventTableTriggerIO 9789: IOValue=[0], IRC5Controller=? -1, Operator=0, SignalSource=ALab_CellC_v1.0_4 5362
EventTableTriggerIO 9790: IOValue=[0], IRC5Controller=? -1, Operator=0, SignalSource=ALab_CellC_v1.0_4 5362
EventTableTriggerIO 9791: IOValue=[1], IRC5Controller=? -1, Operator=0, SignalSource=ALab_CellC_v1.0_4 5362
EventTableTriggerIO 9792: IOValue=[1], IRC5Controller=? -1, Operator=0, SignalSource=ALab_CellC_v1.0_4 5362
EventTableTriggerIO 9793: IOValue=[1], IRC5Controller=? -1, Operator=0, SignalSource=ALab_CellC_v1.0_4 5362
EventTableTriggerIO 9794: IOValue=[1], IRC5Controller=? -1, Operator=0, SignalSource=ALab_CellC_v1.0_4 5362
EventTableTriggerIO 9795: IOValue=[1], IRC5Controller=? -1, Operator=0, SignalSource=ALab_CellC_v1.0_4 5362
EventTableTriggerIO 9796: IOValue=[1], IRC5Controller=? -1, Operator=0, SignalSource=ALab_CellC_v1.0_4 5362
EventTableTriggerIO 9797: IOValue=[1], IRC5Controller=? -1, Operator=0, SignalSource=ALab_CellC_v1.0_4 5362
EventTableTriggerIO 9798: IOValue=[1], IRC5Controller=? -1, Operator=0, SignalSource=ALab_CellC_v1.0_4 5362
EventTableTriggerIO 9799: IOValue=[1], IRC5Controller=? -1, Operator=0, SignalSource=ALab_CellC_v1.0_4 5362
EventTableTriggerIO 9800: IOValue=[1], IRC5Controller=? -1, Operator=0, SignalSource=ALab_CellC_v1.0_4 5362
EventTableTriggerIO 9801: IOValue=[1], IRC5Controller=? -1, Operator=0, SignalSource=ALab_CellC_v1.0_4 5362
EventTableTriggerIO 9802: IOValue=[1], IRC5Controller=? -1, Operator=0, SignalSource=ALab_CellC_v1.0_4 5362
EventTableTriggerIO 9803: IOValue=[0], IRC5Controller=? -1, Operator=0, SignalSource=ALab_CellC_v1.0_4 5362
EventTableTriggerIO 9804: IOValue=[0], IRC5Controller=? -1, Operator=0, SignalSource=ALab_CellC_v1.0_4 5362
EventTableTriggerIO 9805: IOValue=[0], IRC5Controller=? -1, Operator=0, SignalSource=ALab_CellC_v1.0_4 5362
EventTableTriggerIO 9806: IOValue=[0], IRC5Controller=? -1, Operator=0, SignalSource=ALab_CellC_v1.0_4 5362
EventTableTriggerIO 9807: IOValue=[0], IRC5Controller=? -1, Operator=0, SignalSource=ALab_CellC_v1.0_4 5362
EventTableTriggerIO 9808: IOValue=[0], IRC5Controller=? -1, Operator=0, SignalSource=ALab_CellC_v1.0_4 5362
EventTableTriggerIO 9809: IOValue=[1], IRC5Controller=? -1, Operator=0, SignalSource=LCFA_profile 1
EventTableTriggerIO 9810: IOValue=[1], IRC5Controller=? -1, Operator=0, SignalSource=LCFA_profile 1
EventTableTriggerIO 9811: IOValue=[1], IRC5Controller=? -1, Operator=0, SignalSource=LCFA_profile 1
EventTableTriggerIO 9812: IOValue=[1], IRC5Controller=? -1, Operator=0, SignalSource=LCFA_profile 1
EventTableTriggerIO 9813: IOValue=[1], IRC5Controller=? -1, Operator=0, SignalSource=LCFA_profile 1
EventTableTriggerIO 9814: IOValue=[1], IRC5Controller=? -1, Operator=0, SignalSource=LCFA_profile 1
EventTableTriggerIO 9815: IOValue=[1], IRC5Controller=? -1, Operator=0, SignalSource=LCFA_profile 1
EventTableTriggerIO 9816: IOValue=[1], IRC5Controller=? -1, Operator=0, SignalSource=LCFA_profile 1
EventTableTriggerIO 9817: IOValue=[1], IRC5Controller=? -1, Operator=0, SignalSource=LCFA_profile 1
EventTableTriggerIO 9818: IOValue=[1], IRC5Controller=? -1, Operator=0, SignalSource=LCFA_profile 1
EventTableTriggerIO 9819: IOValue=[1], IRC5Controller=? -1, Operator=0, SignalSource=LCFA_profile 1
EventTableTriggerIO 9820: IOValue=[1], IRC5Controller=? -1, Operator=0, SignalSource=LCFA_profile 1
EventTableTriggerIO 9821: IOValue=[1], IRC5Controller=? -1, Operator=0, SignalSource=LCFA_profile 1
EventTableTriggerIO 9822: IOValue=[1], IRC5Controller=? -1, Operator=0, SignalSource=LCFA_profile 1
EventTableTriggerIO 9823: IOValue=[1], IRC5Controller=? -1, Operator=0, SignalSource=LCFA_profile 1
EventTableTriggerIO 9824: IOValue=[1], IRC5Controller=? -1, Operator=0, SignalSource=LCFA_profile 1
EventTableTriggerIO 9825: IOValue=[1], IRC5Controller=? -1, Operator=0, SignalSource=LCFA_profile 1
EventTableTriggerIO 9826: IOValue=[1], IRC5Controller=? -1, Operator=0, SignalSource=LCFA_profile 1
EventTableTriggerLogic 9827: layoutX=150, layoutY=90, Operand1=AND 6770, Operand2=conv2_motor_s1 6766, Operator=0, Delay=1000
EventTableTriggerLogic 9828: layoutX=150, layoutY=90, Operand1=AND 6770, Operand2=conv2_motor_s1 6766, Operator=0, Delay=1000
EventTableTriggerLogic 9829: layoutX=150, layoutY=90, Operand1=AND 6770, Operand2=conv2_motor_s1 6766, Operator=0, Delay=1000
EventTableTriggerLogic 9830: layoutX=150, layoutY=90, Operand1=AND 6770, Operand2=conv2_motor_s1 6766, Operator=0, Delay=1000
EventTableTriggerLogic 9831: layoutX=150, layoutY=90, Operand1=AND 6770, Operand2=conv2_motor_s1 6766, Operator=0, Delay=1000
EventTableTriggerLogic 9832: layoutX=150, layoutY=90, Operand1=AND 6770, Operand2=conv2_motor_s1 6766, Operator=0, Delay=1000
EventTableTriggerIO 9833: IOValue=[1], IRC5Controller=? -1, Operator=0, SignalSource=LCFA_profile 1
EventTableTriggerIO 9834: IOValue=[1], IRC5Controller=? -1, Operator=0, SignalSource=LCFA_profile 1
EventTableTriggerIO 9835: IOValue=[1], IRC5Controller=? -1, Operator=0, SignalSource=LCFA_profile 1
EventTableTriggerIO 9836: IOValue=[1], IRC5Controller=? -1, Operator=0, SignalSource=LCFA_profile 1
EventTableTriggerIO 9837: IOValue=[1], IRC5Controller=? -1, Operator=0, SignalSource=LCFA_profile 1
EventTableTriggerIO 9838: IOValue=[1], IRC5Controller=? -1, Operator=0, SignalSource=LCFA_profile 1
EventTableTriggerIO 9839: IOValue=[1], IRC5Controller=? -1, Operator=0, SignalSource=LCFA_profile 1
EventTableTriggerIO 9840: IOValue=[1], IRC5Controller=? -1, Operator=0, SignalSource=LCFA_profile 1
EventTableTriggerIO 9841: IOValue=[1], IRC5Controller=? -1, Operator=0, SignalSource=LCFA_profile 1
EventTableTriggerIO 9842: IOValue=[1], IRC5Controller=? -1, Operator=0, SignalSource=LCFA_profile 1
EventTableTriggerIO 9843: IOValue=[1], IRC5Controller=? -1, Operator=0, SignalSource=LCFA_profile 1
EventTableTriggerIO 9844: IOValue=[1], IRC5Controller=? -1, Operator=0, SignalSource=LCFA_profile 1
EventTableTriggerIO 9845: IOValue=[1], IRC5Controller=? -1, Operator=0, SignalSource=LCFA_profile 1
EventTableTriggerIO 9846: IOValue=[1], IRC5Controller=? -1, Operator=0, SignalSource=LCFA_profile 1
EventTableTriggerIO 9847: IOValue=[1], IRC5Controller=? -1, Operator=0, SignalSource=LCFA_profile 1
EventTableTriggerIO 9848: IOValue=[1], IRC5Controller=? -1, Operator=0, SignalSource=LCFA_profile 1
EventTableTriggerIO 9849: IOValue=[1], IRC5Controller=? -1, Operator=0, SignalSource=LCFA_profile 1
EventTableTriggerIO 9850: IOValue=[1], IRC5Controller=? -1, Operator=0, SignalSource=LCFA_profile 1
EventTableTriggerIO 9851: IOValue=[1], IRC5Controller=? -1, Operator=0, SignalSource=LCFA_profile 1
EventTableTriggerIO 9852: IOValue=[1], IRC5Controller=? -1, Operator=0, SignalSource=LCFA_profile 1
EventTableTriggerIO 9853: IOValue=[1], IRC5Controller=? -1, Operator=0, SignalSource=LCFA_profile 1
EventTableTriggerIO 9854: IOValue=[1], IRC5Controller=? -1, Operator=0, SignalSource=LCFA_profile 1
EventTableTriggerIO 9855: IOValue=[1], IRC5Controller=? -1, Operator=0, SignalSource=LCFA_profile 1
EventTableTriggerIO 9856: IOValue=[1], IRC5Controller=? -1, Operator=0, SignalSource=LCFA_profile 1
EventTableTriggerIO 9857: IOValue=[1], IRC5Controller=? -1, Operator=0, SignalSource=LCFA_profile 1
EventTableTriggerIO 9858: IOValue=[1], IRC5Controller=? -1, Operator=0, SignalSource=LCFA_profile 1
EventTableTriggerIO 9859: IOValue=[1], IRC5Controller=? -1, Operator=0, SignalSource=LCFA_profile 1
EventTableTriggerIO 9860: IOValue=[1], IRC5Controller=? -1, Operator=0, SignalSource=LCFA_profile 1
EventTableTriggerIO 9861: IOValue=[1], IRC5Controller=? -1, Operator=0, SignalSource=LCFA_profile 1
EventTableTriggerIO 9862: IOValue=[1], IRC5Controller=? -1, Operator=0, SignalSource=LCFA_profile 1
EventTableTriggerIO 9863: IOValue=[1], IRC5Controller=? -1, Operator=0, SignalSource=LCFA_profile 1
EventTableTriggerIO 9864: IOValue=[1], IRC5Controller=? -1, Operator=0, SignalSource=LCFA_profile 1
EventTableTriggerIO 9865: IOValue=[1], IRC5Controller=? -1, Operator=0, SignalSource=LCFA_profile 1
EventTableTriggerIO 9866: IOValue=[1], IRC5Controller=? -1, Operator=0, SignalSource=LCFA_profile 1
EventTableTriggerIO 9867: IOValue=[1], IRC5Controller=? -1, Operator=0, SignalSource=LCFA_profile 1
EventTableTriggerIO 9868: IOValue=[1], IRC5Controller=? -1, Operator=0, SignalSource=LCFA_profile 1
EventTableTriggerIO 9869: IOValue=[1], IRC5Controller=? -1, Operator=0, SignalSource=LCFA_profile 1
EventTableTriggerIO 9870: IOValue=[1], IRC5Controller=? -1, Operator=0, SignalSource=LCFA_profile 1
EventTableTriggerIO 9871: IOValue=[1], IRC5Controller=? -1, Operator=0, SignalSource=LCFA_profile 1
EventTableTriggerIO 9872: IOValue=[1], IRC5Controller=? -1, Operator=0, SignalSource=LCFA_profile 1
EventTableTriggerIO 9873: IOValue=[1], IRC5Controller=? -1, Operator=0, SignalSource=LCFA_profile 1
EventTableTriggerIO 9874: IOValue=[1], IRC5Controller=? -1, Operator=0, SignalSource=LCFA_profile 1
EventTableTriggerIO 9875: IOValue=[1], IRC5Controller=? -1, Operator=0, SignalSource=LCFA_profile 1
EventTableTriggerIO 9876: IOValue=[1], IRC5Controller=? -1, Operator=0, SignalSource=LCFA_profile 1
EventTableTriggerIO 9877: IOValue=[1], IRC5Controller=? -1, Operator=0, SignalSource=LCFA_profile 1
EventTableTriggerIO 9878: IOValue=[1], IRC5Controller=? -1, Operator=0, SignalSource=LCFA_profile 1
EventTableTriggerIO 9879: IOValue=[1], IRC5Controller=? -1, Operator=0, SignalSource=LCFA_profile 1
EventTableTriggerIO 9880: IOValue=[1], IRC5Controller=? -1, Operator=0, SignalSource=LCFA_profile 1
EventTableTriggerIO 9881: IOValue=[1], IRC5Controller=? -1, Operator=0, SignalSource=LCFA_profile 1
EventTableTriggerIO 9882: IOValue=[1], IRC5Controller=? -1, Operator=0, SignalSource=LCFA_profile 1
EventTableTriggerIO 9883: IOValue=[1], IRC5Controller=? -1, Operator=0, SignalSource=LCFA_profile 1
EventTableTriggerIO 9884: IOValue=[1], IRC5Controller=? -1, Operator=0, SignalSource=LCFA_profile 1
EventTableTriggerIO 9885: IOValue=[1], IRC5Controller=? -1, Operator=0, SignalSource=LCFA_profile 1
EventTableTriggerIO 9886: IOValue=[1], IRC5Controller=? -1, Operator=0, SignalSource=LCFA_profile 1
EventTableTriggerIO 9887: IOValue=[1], IRC5Controller=? -1, Operator=0, SignalSource=LCFA_profile 1
EventTableTriggerIO 9888: IOValue=[1], IRC5Controller=? -1, Operator=0, SignalSource=LCFA_profile 1
EventTableTriggerIO 9889: IOValue=[1], IRC5Controller=? -1, Operator=0, SignalSource=LCFA_profile 1
EventTableTriggerIO 9890: IOValue=[1], IRC5Controller=? -1, Operator=0, SignalSource=LCFA_profile 1
EventTableTriggerIO 9891: IOValue=[1], IRC5Controller=? -1, Operator=0, SignalSource=LCFA_profile 1
EventTableTriggerIO 9892: IOValue=[1], IRC5Controller=? -1, Operator=0, SignalSource=LCFA_profile 1
EventTableTriggerIO 9893: IOValue=[1], IRC5Controller=? -1, Operator=0, SignalSource=LCFA_profile 1
EventTableTriggerIO 9894: IOValue=[1], IRC5Controller=? -1, Operator=0, SignalSource=LCFA_profile 1
EventTableTriggerIO 9895: IOValue=[1], IRC5Controller=? -1, Operator=0, SignalSource=LCFA_profile 1
EventTableTriggerIO 9896: IOValue=[1], IRC5Controller=? -1, Operator=0, SignalSource=LCFA_profile 1
EventTableTriggerIO 9897: IOValue=[1], IRC5Controller=? -1, Operator=0, SignalSource=LCFA_profile 1
EventTableTriggerIO 9898: IOValue=[1], IRC5Controller=? -1, Operator=0, SignalSource=LCFA_profile 1
EventTableTriggerIO 9899: IOValue=[1], IRC5Controller=? -1, Operator=0, SignalSource=LCFA_profile 1
EventTableTriggerIO 9900: IOValue=[1], IRC5Controller=? -1, Operator=0, SignalSource=LCFA_profile 1
EventTableTriggerIO 9901: IOValue=[1], IRC5Controller=? -1, Operator=0, SignalSource=LCFA_profile 1
EventTableTriggerIO 9902: IOValue=[1], IRC5Controller=? -1, Operator=0, SignalSource=LCFA_profile 1
EventTableTriggerIO 9903: IOValue=[1], IRC5Controller=? -1, Operator=0, SignalSource=LCFA_profile 1
EventTableTriggerIO 9904: IOValue=[1], IRC5Controller=? -1, Operator=0, SignalSource=LCFA_profile 1
EventTableTriggerLogic 9905: layoutX=155, layoutY=137, Operand1=AND 6751, Operand2=NOT 6755, Operator=0, Delay=1000
EventTableTriggerLogic 9906: layoutX=155, layoutY=137, Operand1=AND 6751, Operand2=NOT 6755, Operator=0, Delay=1000
EventTableTriggerLogic 9907: layoutX=155, layoutY=137, Operand1=AND 6751, Operand2=NOT 6755, Operator=0, Delay=1000
EventTableTriggerLogic 9908: layoutX=155, layoutY=137, Operand1=AND 6751, Operand2=NOT 6755, Operator=0, Delay=1000
EventTableTriggerLogic 9909: layoutX=155, layoutY=137, Operand1=AND 6751, Operand2=NOT 6755, Operator=0, Delay=1000
EventTableTriggerLogic 9910: layoutX=155, layoutY=137, Operand1=AND 6751, Operand2=NOT 6755, Operator=0, Delay=1000
EventTableTriggerIO 9911: IOValue=[1], IRC5Controller=? -1, Operator=0, SignalSource=LCFA_profile 1
EventTableTriggerIO 9912: IOValue=[1], IRC5Controller=? -1, Operator=0, SignalSource=LCFA_profile 1
EventTableTriggerIO 9913: IOValue=[1], IRC5Controller=? -1, Operator=0, SignalSource=LCFA_profile 1
EventTableTriggerIO 9914: IOValue=[1], IRC5Controller=? -1, Operator=0, SignalSource=LCFA_profile 1
EventTableTriggerIO 9915: IOValue=[1], IRC5Controller=? -1, Operator=0, SignalSource=LCFA_profile 1
EventTableTriggerIO 9916: IOValue=[1], IRC5Controller=? -1, Operator=0, SignalSource=LCFA_profile 1
EventTableTriggerIO 9917: IOValue=[1], IRC5Controller=? -1, Operator=0, SignalSource=LCFA_profile 1
EventTableTriggerIO 9918: IOValue=[1], IRC5Controller=? -1, Operator=0, SignalSource=LCFA_profile 1
EventTableTriggerIO 9919: IOValue=[1], IRC5Controller=? -1, Operator=0, SignalSource=LCFA_profile 1
EventTableTriggerIO 9920: IOValue=[1], IRC5Controller=? -1, Operator=0, SignalSource=LCFA_profile 1
EventTableTriggerIO 9921: IOValue=[1], IRC5Controller=? -1, Operator=0, SignalSource=LCFA_profile 1
EventTableTriggerIO 9922: IOValue=[1], IRC5Controller=? -1, Operator=0, SignalSource=LCFA_profile 1
EventTableTriggerLogic 9923: layoutX=48, layoutY=41, Operand1=pallet1.1 6778, Operand2=PalletIO00 6779, Operator=0, Delay=1000
EventTableTriggerLogic 9924: layoutX=48, layoutY=41, Operand1=pallet1.1 6778, Operand2=PalletIO00 6779, Operator=0, Delay=1000
EventTableTriggerLogic 9925: layoutX=48, layoutY=41, Operand1=pallet1.1 6778, Operand2=PalletIO00 6779, Operator=0, Delay=1000
EventTableTriggerLogic 9926: layoutX=48, layoutY=41, Operand1=pallet1.1 6778, Operand2=PalletIO00 6779, Operator=0, Delay=1000
EventTableTriggerLogic 9927: layoutX=48, layoutY=41, Operand1=pallet1.1 6778, Operand2=PalletIO00 6779, Operator=0, Delay=1000
EventTableTriggerLogic 9928: layoutX=48, layoutY=41, Operand1=pallet1.1 6778, Operand2=PalletIO00 6779, Operator=0, Delay=1000
EventTableTriggerIO 9929: IOValue=[1], IRC5Controller=? -1, Operator=0, SignalSource=LCFA_profile 1
EventTableTriggerIO 9930: IOValue=[1], IRC5Controller=? -1, Operator=0, SignalSource=LCFA_profile 1
EventTableTriggerIO 9931: IOValue=[1], IRC5Controller=? -1, Operator=0, SignalSource=LCFA_profile 1
EventTableTriggerIO 9932: IOValue=[1], IRC5Controller=? -1, Operator=0, SignalSource=LCFA_profile 1
EventTableTriggerIO 9933: IOValue=[1], IRC5Controller=? -1, Operator=0, SignalSource=LCFA_profile 1
EventTableTriggerIO 9934: IOValue=[1], IRC5Controller=? -1, Operator=0, SignalSource=LCFA_profile 1
EventTableTriggerIO 9935: IOValue=[1], IRC5Controller=? -1, Operator=0, SignalSource=ALab_CellC_v1.0_4 5362
EventTableTriggerIO 9936: IOValue=[1], IRC5Controller=? -1, Operator=0, SignalSource=ALab_CellC_v1.0_4 5362
EventTableTriggerIO 9937: IOValue=[1], IRC5Controller=? -1, Operator=0, SignalSource=ALab_CellC_v1.0_4 5362
EventTableTriggerIO 9938: IOValue=[1], IRC5Controller=? -1, Operator=0, SignalSource=ALab_CellC_v1.0_4 5362
EventTableTriggerIO 9939: IOValue=[1], IRC5Controller=? -1, Operator=0, SignalSource=ALab_CellC_v1.0_4 5362
EventTableTriggerIO 9940: IOValue=[1], IRC5Controller=? -1, Operator=0, SignalSource=ALab_CellC_v1.0_4 5362
EventTableTriggerIO 9941: IOValue=[0], IRC5Controller=? -1, Operator=0, SignalSource=ALab_CellC_v1.0_4 5362
EventTableTriggerIO 9942: IOValue=[0], IRC5Controller=? -1, Operator=0, SignalSource=ALab_CellC_v1.0_4 5362
EventTableTriggerIO 9943: IOValue=[0], IRC5Controller=? -1, Operator=0, SignalSource=ALab_CellC_v1.0_4 5362
EventTableTriggerIO 9944: IOValue=[0], IRC5Controller=? -1, Operator=0, SignalSource=ALab_CellC_v1.0_4 5362
EventTableTriggerIO 9945: IOValue=[0], IRC5Controller=? -1, Operator=0, SignalSource=ALab_CellC_v1.0_4 5362
EventTableTriggerIO 9946: IOValue=[0], IRC5Controller=? -1, Operator=0, SignalSource=ALab_CellC_v1.0_4 5362
EventTableTriggerLogic 9947: layoutX=103, layoutY=47, Operand1=NOT 8291, Operand2=pallet5 8290, Operator=0, Delay=1000
EventTableTriggerLogic 9948: layoutX=103, layoutY=47, Operand1=NOT 8291, Operand2=pallet5 8290, Operator=0, Delay=1000
EventTableTriggerLogic 9949: layoutX=103, layoutY=47, Operand1=NOT 8291, Operand2=pallet5 8290, Operator=0, Delay=1000
EventTableTriggerLogic 9950: layoutX=103, layoutY=47, Operand1=NOT 8291, Operand2=pallet5 8290, Operator=0, Delay=1000
EventTableTriggerLogic 9951: layoutX=103, layoutY=47, Operand1=NOT 8291, Operand2=pallet5 8290, Operator=0, Delay=1000
EventTableTriggerLogic 9952: layoutX=103, layoutY=47, Operand1=NOT 8291, Operand2=pallet5 8290, Operator=0, Delay=1000
EventTableTriggerLogic 9953: layoutX=79, layoutY=37, Operand1=Pallet5.3 8029, Operand2=conv2_buffer_upper_vertical_move 8133, Operator=0, Delay=1000
EventTableTriggerLogic 9954: layoutX=79, layoutY=37, Operand1=Pallet5.3 8029, Operand2=conv2_buffer_upper_vertical_move 8133, Operator=0, Delay=1000
EventTableTriggerLogic 9955: layoutX=79, layoutY=37, Operand1=Pallet5.3 8029, Operand2=conv2_buffer_upper_vertical_move 8133, Operator=0, Delay=1000
EventTableTriggerLogic 9956: layoutX=79, layoutY=37, Operand1=Pallet5.3 8029, Operand2=conv2_buffer_upper_vertical_move 8133, Operator=0, Delay=1000
EventTableTriggerLogic 9957: layoutX=79, layoutY=37, Operand1=Pallet5.3 8029, Operand2=conv2_buffer_upper_vertical_move 8133, Operator=0, Delay=1000
EventTableTriggerLogic 9958: layoutX=79, layoutY=37, Operand1=Pallet5.3 8029, Operand2=conv2_buffer_upper_vertical_move 8133, Operator=0, Delay=1000
EventTableTriggerLogic 9959: layoutX=40, layoutY=37, Operand1=Pallet5.4 8035, Operand2=conv2_buffer_lower_vertical_move 8036, Operator=0, Delay=1000
EventTableTriggerLogic 9960: layoutX=40, layoutY=37, Operand1=Pallet5.4 8035, Operand2=conv2_buffer_lower_vertical_move 8036, Operator=0, Delay=1000
EventTableTriggerLogic 9961: layoutX=40, layoutY=37, Operand1=Pallet5.4 8035, Operand2=conv2_buffer_lower_vertical_move 8036, Operator=0, Delay=1000
EventTableTriggerLogic 9962: layoutX=40, layoutY=37, Operand1=Pallet5.4 8035, Operand2=conv2_buffer_lower_vertical_move 8036, Operator=0, Delay=1000
EventTableTriggerLogic 9963: layoutX=40, layoutY=37, Operand1=Pallet5.4 8035, Operand2=conv2_buffer_lower_vertical_move 8036, Operator=0, Delay=1000
EventTableTriggerLogic 9964: layoutX=40, layoutY=37, Operand1=Pallet5.4 8035, Operand2=conv2_buffer_lower_vertical_move 8036, Operator=0, Delay=1000
EventTableTriggerLogic 9965: layoutX=103, layoutY=47, Operand1=conv2_buffer_horizontal_move 8134, Operand2=Pallet5.7 8040, Operator=0, Delay=1000
EventTableTriggerLogic 9966: layoutX=103, layoutY=47, Operand1=conv2_buffer_horizontal_move 8134, Operand2=Pallet5.7 8040, Operator=0, Delay=1000
EventTableTriggerLogic 9967: layoutX=103, layoutY=47, Operand1=conv2_buffer_horizontal_move 8134, Operand2=Pallet5.7 8040, Operator=0, Delay=1000
EventTableTriggerLogic 9968: layoutX=103, layoutY=47, Operand1=conv2_buffer_horizontal_move 8134, Operand2=Pallet5.7 8040, Operator=0, Delay=1000
EventTableTriggerLogic 9969: layoutX=103, layoutY=47, Operand1=conv2_buffer_horizontal_move 8134, Operand2=Pallet5.7 8040, Operator=0, Delay=1000
EventTableTriggerLogic 9970: layoutX=103, layoutY=47, Operand1=conv2_buffer_horizontal_move 8134, Operand2=Pallet5.7 8040, Operator=0, Delay=1000
EventTableTriggerLogic 9971: layoutX=54, layoutY=45, Operand1=NOT 8135, Operand2=Pallet5.6 8046, Operator=0, Delay=1000
EventTableTriggerLogic 9972: layoutX=54, layoutY=45, Operand1=NOT 8135, Operand2=Pallet5.6 8046, Operator=0, Delay=1000
EventTableTriggerLogic 9973: layoutX=54, layoutY=45, Operand1=NOT 8135, Operand2=Pallet5.6 8046, Operator=0, Delay=1000
EventTableTriggerLogic 9974: layoutX=54, layoutY=45, Operand1=NOT 8135, Operand2=Pallet5.6 8046, Operator=0, Delay=1000
EventTableTriggerLogic 9975: layoutX=54, layoutY=45, Operand1=NOT 8135, Operand2=Pallet5.6 8046, Operator=0, Delay=1000
EventTableTriggerLogic 9976: layoutX=54, layoutY=45, Operand1=NOT 8135, Operand2=Pallet5.6 8046, Operator=0, Delay=1000
EventTableTriggerLogic 9977: layoutX=108, layoutY=46, Operand1=NOT 8052, Operand2=Pallet5.5 8051, Operator=0, Delay=1000
EventTableTriggerLogic 9978: layoutX=108, layoutY=46, Operand1=NOT 8052, Operand2=Pallet5.5 8051, Operator=0, Delay=1000
EventTableTriggerLogic 9979: layoutX=108, layoutY=46, Operand1=NOT 8052, Operand2=Pallet5.5 8051, Operator=0, Delay=1000
EventTableTriggerLogic 9980: layoutX=108, layoutY=46, Operand1=NOT 8052, Operand2=Pallet5.5 8051, Operator=0, Delay=1000
EventTableTriggerLogic 9981: layoutX=108, layoutY=46, Operand1=NOT 8052, Operand2=Pallet5.5 8051, Operator=0, Delay=1000
EventTableTriggerLogic 9982: layoutX=108, layoutY=46, Operand1=NOT 8052, Operand2=Pallet5.5 8051, Operator=0, Delay=1000
EventTableTriggerIO 9983: IOValue=[1], IRC5Controller=? -1, Operator=0, SignalSource=LCFA_profile 1
EventTableTriggerIO 9984: IOValue=[1], IRC5Controller=? -1, Operator=0, SignalSource=LCFA_profile 1
EventTableTriggerIO 9985: IOValue=[1], IRC5Controller=? -1, Operator=0, SignalSource=LCFA_profile 1
EventTableTriggerIO 9986: IOValue=[1], IRC5Controller=? -1, Operator=0, SignalSource=LCFA_profile 1
EventTableTriggerIO 9987: IOValue=[1], IRC5Controller=? -1, Operator=0, SignalSource=LCFA_profile 1
EventTableTriggerIO 9988: IOValue=[1], IRC5Controller=? -1, Operator=0, SignalSource=LCFA_profile 1
EventTableTriggerIO 9989: IOValue=[1], IRC5Controller=? -1, Operator=0, SignalSource=LCFA_profile 1
EventTableTriggerIO 9990: IOValue=[1], IRC5Controller=? -1, Operator=0, SignalSource=LCFA_profile 1
EventTableTriggerIO 9991: IOValue=[1], IRC5Controller=? -1, Operator=0, SignalSource=LCFA_profile 1
EventTableTriggerIO 9992: IOValue=[1], IRC5Controller=? -1, Operator=0, SignalSource=LCFA_profile 1
EventTableTriggerIO 9993: IOValue=[1], IRC5Controller=? -1, Operator=0, SignalSource=LCFA_profile 1
EventTableTriggerIO 9994: IOValue=[1], IRC5Controller=? -1, Operator=0, SignalSource=LCFA_profile 1
EventTableTriggerIO 9995: IOValue=[1], IRC5Controller=? -1, Operator=0, SignalSource=LCFA_profile 1
EventTableTriggerIO 9996: IOValue=[1], IRC5Controller=? -1, Operator=0, SignalSource=LCFA_profile 1
EventTableTriggerIO 9997: IOValue=[1], IRC5Controller=? -1, Operator=0, SignalSource=LCFA_profile 1
EventTableTriggerIO 9998: IOValue=[1], IRC5Controller=? -1, Operator=0, SignalSource=LCFA_profile 1
EventTableTriggerIO 9999: IOValue=[1], IRC5Controller=? -1, Operator=0, SignalSource=LCFA_profile 1
EventTableTriggerIO 10000: IOValue=[1], IRC5Controller=? -1, Operator=0, SignalSource=LCFA_profile 1
EventTableTriggerIO 10001: IOValue=[1], IRC5Controller=? -1, Operator=0, SignalSource=LCFA_profile 1
EventTableTriggerIO 10002: IOValue=[1], IRC5Controller=? -1, Operator=0, SignalSource=LCFA_profile 1
EventTableTriggerIO 10003: IOValue=[1], IRC5Controller=? -1, Operator=0, SignalSource=LCFA_profile 1
EventTableTriggerIO 10004: IOValue=[1], IRC5Controller=? -1, Operator=0, SignalSource=LCFA_profile 1
EventTableTriggerIO 10005: IOValue=[1], IRC5Controller=? -1, Operator=0, SignalSource=LCFA_profile 1
EventTableTriggerIO 10006: IOValue=[1], IRC5Controller=? -1, Operator=0, SignalSource=LCFA_profile 1
EventTableTriggerIO 10007: IOValue=[1], IRC5Controller=? -1, Operator=0, SignalSource=LCFA_profile 1
EventTableTriggerIO 10008: IOValue=[1], IRC5Controller=? -1, Operator=0, SignalSource=LCFA_profile 1
EventTableTriggerIO 10009: IOValue=[1], IRC5Controller=? -1, Operator=0, SignalSource=LCFA_profile 1
EventTableTriggerIO 10010: IOValue=[1], IRC5Controller=? -1, Operator=0, SignalSource=LCFA_profile 1
EventTableTriggerIO 10011: IOValue=[1], IRC5Controller=? -1, Operator=0, SignalSource=LCFA_profile 1
EventTableTriggerIO 10012: IOValue=[1], IRC5Controller=? -1, Operator=0, SignalSource=LCFA_profile 1
EventTableTriggerIO 10013: IOValue=[1], IRC5Controller=? -1, Operator=0, SignalSource=LCFA_profile 1
EventTableTriggerIO 10014: IOValue=[1], IRC5Controller=? -1, Operator=0, SignalSource=LCFA_profile 1
EventTableTriggerIO 10015: IOValue=[1], IRC5Controller=? -1, Operator=0, SignalSource=LCFA_profile 1
EventTableTriggerIO 10016: IOValue=[1], IRC5Controller=? -1, Operator=0, SignalSource=LCFA_profile 1
EventTableTriggerIO 10017: IOValue=[1], IRC5Controller=? -1, Operator=0, SignalSource=LCFA_profile 1
EventTableTriggerIO 10018: IOValue=[1], IRC5Controller=? -1, Operator=0, SignalSource=LCFA_profile 1
EventTableTriggerIO 10019: IOValue=[1], IRC5Controller=? -1, Operator=0, SignalSource=LCFA_profile 1
EventTableTriggerIO 10020: IOValue=[1], IRC5Controller=? -1, Operator=0, SignalSource=LCFA_profile 1
EventTableTriggerIO 10021: IOValue=[1], IRC5Controller=? -1, Operator=0, SignalSource=LCFA_profile 1
EventTableTriggerIO 10022: IOValue=[1], IRC5Controller=? -1, Operator=0, SignalSource=LCFA_profile 1
EventTableTriggerIO 10023: IOValue=[1], IRC5Controller=? -1, Operator=0, SignalSource=LCFA_profile 1
EventTableTriggerIO 10024: IOValue=[1], IRC5Controller=? -1, Operator=0, SignalSource=LCFA_profile 1
EventTableTriggerIO 10025: IOValue=[1], IRC5Controller=? -1, Operator=0, SignalSource=LCFA_profile 1
EventTableTriggerIO 10026: IOValue=[1], IRC5Controller=? -1, Operator=0, SignalSource=LCFA_profile 1
EventTableTriggerIO 10027: IOValue=[1], IRC5Controller=? -1, Operator=0, SignalSource=LCFA_profile 1
EventTableTriggerIO 10028: IOValue=[1], IRC5Controller=? -1, Operator=0, SignalSource=LCFA_profile 1
EventTableTriggerIO 10029: IOValue=[1], IRC5Controller=? -1, Operator=0, SignalSource=LCFA_profile 1
EventTableTriggerIO 10030: IOValue=[1], IRC5Controller=? -1, Operator=0, SignalSource=LCFA_profile 1
EventTableTriggerIO 10031: IOValue=[1], IRC5Controller=? -1, Operator=0, SignalSource=LCFA_profile 1
EventTableTriggerIO 10032: IOValue=[1], IRC5Controller=? -1, Operator=0, SignalSource=LCFA_profile 1
EventTableTriggerIO 10033: IOValue=[1], IRC5Controller=? -1, Operator=0, SignalSource=LCFA_profile 1
EventTableTriggerIO 10034: IOValue=[1], IRC5Controller=? -1, Operator=0, SignalSource=LCFA_profile 1
EventTableTriggerIO 10035: IOValue=[1], IRC5Controller=? -1, Operator=0, SignalSource=LCFA_profile 1
EventTableTriggerIO 10036: IOValue=[1], IRC5Controller=? -1, Operator=0, SignalSource=LCFA_profile 1
EventTableTriggerIO 10037: IOValue=[1], IRC5Controller=? -1, Operator=0, SignalSource=LCFA_profile 1
EventTableTriggerIO 10038: IOValue=[1], IRC5Controller=? -1, Operator=0, SignalSource=LCFA_profile 1
EventTableTriggerIO 10039: IOValue=[1], IRC5Controller=? -1, Operator=0, SignalSource=LCFA_profile 1
EventTableTriggerIO 10040: IOValue=[1], IRC5Controller=? -1, Operator=0, SignalSource=LCFA_profile 1
EventTableTriggerIO 10041: IOValue=[1], IRC5Controller=? -1, Operator=0, SignalSource=LCFA_profile 1
EventTableTriggerIO 10042: IOValue=[1], IRC5Controller=? -1, Operator=0, SignalSource=LCFA_profile 1
EventTableTriggerIO 10043: IOValue=[1], IRC5Controller=? -1, Operator=0, SignalSource=LCFA_profile 1
EventTableTriggerIO 10044: IOValue=[1], IRC5Controller=? -1, Operator=0, SignalSource=LCFA_profile 1
EventTableTriggerIO 10045: IOValue=[1], IRC5Controller=? -1, Operator=0, SignalSource=LCFA_profile 1
EventTableTriggerIO 10046: IOValue=[1], IRC5Controller=? -1, Operator=0, SignalSource=LCFA_profile 1
EventTableTriggerIO 10047: IOValue=[1], IRC5Controller=? -1, Operator=0, SignalSource=LCFA_profile 1
EventTableTriggerIO 10048: IOValue=[1], IRC5Controller=? -1, Operator=0, SignalSource=LCFA_profile 1
EventTableTriggerIO 10049: IOValue=[1], IRC5Controller=? -1, Operator=0, SignalSource=LCFA_profile 1
EventTableTriggerIO 10050: IOValue=[1], IRC5Controller=? -1, Operator=0, SignalSource=LCFA_profile 1
EventTableTriggerIO 10051: IOValue=[1], IRC5Controller=? -1, Operator=0, SignalSource=LCFA_profile 1
EventTableTriggerIO 10052: IOValue=[1], IRC5Controller=? -1, Operator=0, SignalSource=LCFA_profile 1
EventTableTriggerIO 10053: IOValue=[1], IRC5Controller=? -1, Operator=0, SignalSource=LCFA_profile 1
EventTableTriggerIO 10054: IOValue=[1], IRC5Controller=? -1, Operator=0, SignalSource=LCFA_profile 1
EventTableTriggerIO 10055: IOValue=[1], IRC5Controller=? -1, Operator=0, SignalSource=LCFA_profile 1
EventTableTriggerIO 10056: IOValue=[1], IRC5Controller=? -1, Operator=0, SignalSource=LCFA_profile 1
EventTableTriggerIO 10057: IOValue=[1], IRC5Controller=? -1, Operator=0, SignalSource=LCFA_profile 1
EventTableTriggerIO 10058: IOValue=[1], IRC5Controller=? -1, Operator=0, SignalSource=LCFA_profile 1
EventTableTriggerIO 10059: IOValue=[1], IRC5Controller=? -1, Operator=0, SignalSource=LCFA_profile 1
EventTableTriggerIO 10060: IOValue=[1], IRC5Controller=? -1, Operator=0, SignalSource=LCFA_profile 1
EventTableTriggerIO 10061: IOValue=[1], IRC5Controller=? -1, Operator=0, SignalSource=LCFA_profile 1
EventTableTriggerIO 10062: IOValue=[1], IRC5Controller=? -1, Operator=0, SignalSource=LCFA_profile 1
EventTableTriggerIO 10063: IOValue=[1], IRC5Controller=? -1, Operator=0, SignalSource=LCFA_profile 1
EventTableTriggerIO 10064: IOValue=[1], IRC5Controller=? -1, Operator=0, SignalSource=LCFA_profile 1
EventTableTriggerIO 10065: IOValue=[1], IRC5Controller=? -1, Operator=0, SignalSource=LCFA_profile 1
EventTableTriggerIO 10066: IOValue=[1], IRC5Controller=? -1, Operator=0, SignalSource=LCFA_profile 1
EventTableTriggerIO 10067: IOValue=[1], IRC5Controller=? -1, Operator=0, SignalSource=LCFA_profile 1
EventTableTriggerIO 10068: IOValue=[1], IRC5Controller=? -1, Operator=0, SignalSource=LCFA_profile 1
EventTableTriggerIO 10069: IOValue=[1], IRC5Controller=? -1, Operator=0, SignalSource=LCFA_profile 1
EventTableTriggerIO 10070: IOValue=[1], IRC5Controller=? -1, Operator=0, SignalSource=LCFA_profile 1
EventTableTriggerIO 10071: IOValue=[1], IRC5Controller=? -1, Operator=0, SignalSource=LCFA_profile 1
EventTableTriggerIO 10072: IOValue=[1], IRC5Controller=? -1, Operator=0, SignalSource=LCFA_profile 1
EventTableTriggerIO 10073: IOValue=[1], IRC5Controller=? -1, Operator=0, SignalSource=LCFA_profile 1
EventTableTriggerIO 10074: IOValue=[1], IRC5Controller=? -1, Operator=0, SignalSource=LCFA_profile 1
EventTableTriggerIO 10075: IOValue=[1], IRC5Controller=? -1, Operator=0, SignalSource=LCFA_profile 1
EventTableTriggerIO 10076: IOValue=[1], IRC5Controller=? -1, Operator=0, SignalSource=LCFA_profile 1
EventTableTriggerIO 10077: IOValue=[1], IRC5Controller=? -1, Operator=0, SignalSource=LCFA_profile 1
EventTableTriggerIO 10078: IOValue=[1], IRC5Controller=? -1, Operator=0, SignalSource=LCFA_profile 1
EventTableTriggerIO 10079: IOValue=[1], IRC5Controller=? -1, Operator=0, SignalSource=LCFA_profile 1
EventTableTriggerIO 10080: IOValue=[1], IRC5Controller=? -1, Operator=0, SignalSource=LCFA_profile 1
EventTableTriggerIO 10081: IOValue=[1], IRC5Controller=? -1, Operator=0, SignalSource=LCFA_profile 1
EventTableTriggerIO 10082: IOValue=[1], IRC5Controller=? -1, Operator=0, SignalSource=LCFA_profile 1
EventTableTriggerIO 10083: IOValue=[1], IRC5Controller=? -1, Operator=0, SignalSource=LCFA_profile 1
EventTableTriggerIO 10084: IOValue=[1], IRC5Controller=? -1, Operator=0, SignalSource=LCFA_profile 1
EventTableTriggerLogic 10085: layoutX=99, layoutY=32, Operand1=Pallet2.1 8141, Operand2=NOT 8139, Operator=0, Delay=1000
EventTableTriggerLogic 10086: layoutX=99, layoutY=32, Operand1=Pallet2.1 8141, Operand2=NOT 8139, Operator=0, Delay=1000
EventTableTriggerLogic 10087: layoutX=99, layoutY=32, Operand1=Pallet2.1 8141, Operand2=NOT 8139, Operator=0, Delay=1000
EventTableTriggerLogic 10088: layoutX=99, layoutY=32, Operand1=Pallet2.1 8141, Operand2=NOT 8139, Operator=0, Delay=1000
EventTableTriggerLogic 10089: layoutX=99, layoutY=32, Operand1=Pallet2.1 8141, Operand2=NOT 8139, Operator=0, Delay=1000
EventTableTriggerLogic 10090: layoutX=99, layoutY=32, Operand1=Pallet2.1 8141, Operand2=NOT 8139, Operator=0, Delay=1000
EventTableTriggerLogic 10091: layoutX=181, layoutY=52, Operand1=conv1_buffer_upper_go_down 8146, Operand2=Pallet2.2 8145, Operator=0, Delay=1000
EventTableTriggerLogic 10092: layoutX=181, layoutY=52, Operand1=conv1_buffer_upper_go_down 8146, Operand2=Pallet2.2 8145, Operator=0, Delay=1000
EventTableTriggerLogic 10093: layoutX=181, layoutY=52, Operand1=conv1_buffer_upper_go_down 8146, Operand2=Pallet2.2 8145, Operator=0, Delay=1000
EventTableTriggerLogic 10094: layoutX=181, layoutY=52, Operand1=conv1_buffer_upper_go_down 8146, Operand2=Pallet2.2 8145, Operator=0, Delay=1000
EventTableTriggerLogic 10095: layoutX=181, layoutY=52, Operand1=conv1_buffer_upper_go_down 8146, Operand2=Pallet2.2 8145, Operator=0, Delay=1000
EventTableTriggerLogic 10096: layoutX=181, layoutY=52, Operand1=conv1_buffer_upper_go_down 8146, Operand2=Pallet2.2 8145, Operator=0, Delay=1000
EventTableTriggerLogic 10097: layoutX=48, layoutY=51, Operand1=Pallet2.3 8150, Operand2=conv1_buffer_lower_go_up 8151, Operator=0, Delay=1000
EventTableTriggerLogic 10098: layoutX=48, layoutY=51, Operand1=Pallet2.3 8150, Operand2=conv1_buffer_lower_go_up 8151, Operator=0, Delay=1000
EventTableTriggerLogic 10099: layoutX=48, layoutY=51, Operand1=Pallet2.3 8150, Operand2=conv1_buffer_lower_go_up 8151, Operator=0, Delay=1000
EventTableTriggerLogic 10100: layoutX=48, layoutY=51, Operand1=Pallet2.3 8150, Operand2=conv1_buffer_lower_go_up 8151, Operator=0, Delay=1000
EventTableTriggerLogic 10101: layoutX=48, layoutY=51, Operand1=Pallet2.3 8150, Operand2=conv1_buffer_lower_go_up 8151, Operator=0, Delay=1000
EventTableTriggerLogic 10102: layoutX=48, layoutY=51, Operand1=Pallet2.3 8150, Operand2=conv1_buffer_lower_go_up 8151, Operator=0, Delay=1000
EventTableTriggerLogic 10103: layoutX=67, layoutY=33, Operand1=pallet2 8155, Operand2=NOT 8156, Operator=0, Delay=1000
EventTableTriggerLogic 10104: layoutX=67, layoutY=33, Operand1=pallet2 8155, Operand2=NOT 8156, Operator=0, Delay=1000
EventTableTriggerLogic 10105: layoutX=67, layoutY=33, Operand1=pallet2 8155, Operand2=NOT 8156, Operator=0, Delay=1000
EventTableTriggerLogic 10106: layoutX=67, layoutY=33, Operand1=pallet2 8155, Operand2=NOT 8156, Operator=0, Delay=1000
EventTableTriggerLogic 10107: layoutX=67, layoutY=33, Operand1=pallet2 8155, Operand2=NOT 8156, Operator=0, Delay=1000
EventTableTriggerLogic 10108: layoutX=67, layoutY=33, Operand1=pallet2 8155, Operand2=NOT 8156, Operator=0, Delay=1000
EventTableTriggerLogic 10109: layoutX=102, layoutY=29, Operand1=Pallet2.4 8161, Operand2=NOT 8162, Operator=0, Delay=1000
EventTableTriggerLogic 10110: layoutX=102, layoutY=29, Operand1=Pallet2.4 8161, Operand2=NOT 8162, Operator=0, Delay=1000
EventTableTriggerLogic 10111: layoutX=102, layoutY=29, Operand1=Pallet2.4 8161, Operand2=NOT 8162, Operator=0, Delay=1000
EventTableTriggerLogic 10112: layoutX=102, layoutY=29, Operand1=Pallet2.4 8161, Operand2=NOT 8162, Operator=0, Delay=1000
EventTableTriggerLogic 10113: layoutX=102, layoutY=29, Operand1=Pallet2.4 8161, Operand2=NOT 8162, Operator=0, Delay=1000
EventTableTriggerLogic 10114: layoutX=102, layoutY=29, Operand1=Pallet2.4 8161, Operand2=NOT 8162, Operator=0, Delay=1000
EventTableTriggerLogic 10115: layoutX=102, layoutY=23, Operand1=Pallet2.5 8167, Operand2=NOT 8168, Operator=0, Delay=1000
EventTableTriggerLogic 10116: layoutX=102, layoutY=23, Operand1=Pallet2.5 8167, Operand2=NOT 8168, Operator=0, Delay=1000
EventTableTriggerLogic 10117: layoutX=102, layoutY=23, Operand1=Pallet2.5 8167, Operand2=NOT 8168, Operator=0, Delay=1000
EventTableTriggerLogic 10118: layoutX=102, layoutY=23, Operand1=Pallet2.5 8167, Operand2=NOT 8168, Operator=0, Delay=1000
EventTableTriggerLogic 10119: layoutX=102, layoutY=23, Operand1=Pallet2.5 8167, Operand2=NOT 8168, Operator=0, Delay=1000
EventTableTriggerLogic 10120: layoutX=102, layoutY=23, Operand1=Pallet2.5 8167, Operand2=NOT 8168, Operator=0, Delay=1000
EventTableTriggerIO 10121: IOValue=[1], IRC5Controller=? -1, Operator=0, SignalSource=LCFA_profile 1
EventTableTriggerIO 10122: IOValue=[1], IRC5Controller=? -1, Operator=0, SignalSource=LCFA_profile 1
EventTableTriggerIO 10123: IOValue=[1], IRC5Controller=? -1, Operator=0, SignalSource=LCFA_profile 1
EventTableTriggerIO 10124: IOValue=[1], IRC5Controller=? -1, Operator=0, SignalSource=LCFA_profile 1
EventTableTriggerIO 10125: IOValue=[1], IRC5Controller=? -1, Operator=0, SignalSource=LCFA_profile 1
EventTableTriggerIO 10126: IOValue=[1], IRC5Controller=? -1, Operator=0, SignalSource=LCFA_profile 1
EventTableTriggerIO 10127: IOValue=[1], IRC5Controller=? -1, Operator=0, SignalSource=LCFA_profile 1
EventTableTriggerIO 10128: IOValue=[1], IRC5Controller=? -1, Operator=0, SignalSource=LCFA_profile 1
EventTableTriggerIO 10129: IOValue=[1], IRC5Controller=? -1, Operator=0, SignalSource=LCFA_profile 1
EventTableTriggerIO 10130: IOValue=[1], IRC5Controller=? -1, Operator=0, SignalSource=LCFA_profile 1
EventTableTriggerIO 10131: IOValue=[1], IRC5Controller=? -1, Operator=0, SignalSource=LCFA_profile 1
EventTableTriggerIO 10132: IOValue=[1], IRC5Controller=? -1, Operator=0, SignalSource=LCFA_profile 1
EventTableTriggerIO 10133: IOValue=[1], IRC5Controller=? -1, Operator=0, SignalSource=LCFA_profile 1
EventTableTriggerIO 10134: IOValue=[1], IRC5Controller=? -1, Operator=0, SignalSource=LCFA_profile 1
EventTableTriggerIO 10135: IOValue=[1], IRC5Controller=? -1, Operator=0, SignalSource=LCFA_profile 1
EventTableTriggerIO 10136: IOValue=[1], IRC5Controller=? -1, Operator=0, SignalSource=LCFA_profile 1
EventTableTriggerIO 10137: IOValue=[1], IRC5Controller=? -1, Operator=0, SignalSource=LCFA_profile 1
EventTableTriggerIO 10138: IOValue=[1], IRC5Controller=? -1, Operator=0, SignalSource=LCFA_profile 1
EventTableTriggerIO 10139: IOValue=[1], IRC5Controller=? -1, Operator=0, SignalSource=LCFA_profile 1
EventTableTriggerIO 10140: IOValue=[1], IRC5Controller=? -1, Operator=0, SignalSource=LCFA_profile 1
EventTableTriggerIO 10141: IOValue=[1], IRC5Controller=? -1, Operator=0, SignalSource=LCFA_profile 1
EventTableTriggerIO 10142: IOValue=[1], IRC5Controller=? -1, Operator=0, SignalSource=LCFA_profile 1
EventTableTriggerIO 10143: IOValue=[1], IRC5Controller=? -1, Operator=0, SignalSource=LCFA_profile 1
EventTableTriggerIO 10144: IOValue=[1], IRC5Controller=? -1, Operator=0, SignalSource=LCFA_profile 1
EventTableTriggerIO 10145: IOValue=[1], IRC5Controller=? -1, Operator=0, SignalSource=LCFA_profile 1
EventTableTriggerIO 10146: IOValue=[1], IRC5Controller=? -1, Operator=0, SignalSource=LCFA_profile 1
EventTableTriggerIO 10147: IOValue=[1], IRC5Controller=? -1, Operator=0, SignalSource=LCFA_profile 1
EventTableTriggerIO 10148: IOValue=[1], IRC5Controller=? -1, Operator=0, SignalSource=LCFA_profile 1
EventTableTriggerIO 10149: IOValue=[1], IRC5Controller=? -1, Operator=0, SignalSource=LCFA_profile 1
EventTableTriggerIO 10150: IOValue=[1], IRC5Controller=? -1, Operator=0, SignalSource=LCFA_profile 1
EventTableTriggerIO 10151: IOValue=[1], IRC5Controller=? -1, Operator=0, SignalSource=LCFA_profile 1
EventTableTriggerIO 10152: IOValue=[1], IRC5Controller=? -1, Operator=0, SignalSource=LCFA_profile 1
EventTableTriggerIO 10153: IOValue=[1], IRC5Controller=? -1, Operator=0, SignalSource=LCFA_profile 1
EventTableTriggerIO 10154: IOValue=[1], IRC5Controller=? -1, Operator=0, SignalSource=LCFA_profile 1
EventTableTriggerIO 10155: IOValue=[1], IRC5Controller=? -1, Operator=0, SignalSource=LCFA_profile 1
EventTableTriggerIO 10156: IOValue=[1], IRC5Controller=? -1, Operator=0, SignalSource=LCFA_profile 1
EventTableTriggerIO 10157: IOValue=[1], IRC5Controller=? -1, Operator=0, SignalSource=LCFA_profile 1
EventTableTriggerIO 10158: IOValue=[1], IRC5Controller=? -1, Operator=0, SignalSource=LCFA_profile 1
EventTableTriggerIO 10159: IOValue=[1], IRC5Controller=? -1, Operator=0, SignalSource=LCFA_profile 1
EventTableTriggerIO 10160: IOValue=[1], IRC5Controller=? -1, Operator=0, SignalSource=LCFA_profile 1
EventTableTriggerIO 10161: IOValue=[1], IRC5Controller=? -1, Operator=0, SignalSource=LCFA_profile 1
EventTableTriggerIO 10162: IOValue=[1], IRC5Controller=? -1, Operator=0, SignalSource=LCFA_profile 1
EventTableTriggerIO 10163: IOValue=[1], IRC5Controller=? -1, Operator=0, SignalSource=LCFA_profile 1
EventTableTriggerIO 10164: IOValue=[1], IRC5Controller=? -1, Operator=0, SignalSource=LCFA_profile 1
EventTableTriggerIO 10165: IOValue=[1], IRC5Controller=? -1, Operator=0, SignalSource=LCFA_profile 1
EventTableTriggerIO 10166: IOValue=[1], IRC5Controller=? -1, Operator=0, SignalSource=LCFA_profile 1
EventTableTriggerIO 10167: IOValue=[1], IRC5Controller=? -1, Operator=0, SignalSource=LCFA_profile 1
EventTableTriggerIO 10168: IOValue=[1], IRC5Controller=? -1, Operator=0, SignalSource=LCFA_profile 1
EventTableTriggerIO 10169: IOValue=[1], IRC5Controller=? -1, Operator=0, SignalSource=LCFA_profile 1
EventTableTriggerIO 10170: IOValue=[1], IRC5Controller=? -1, Operator=0, SignalSource=LCFA_profile 1
EventTableTriggerIO 10171: IOValue=[1], IRC5Controller=? -1, Operator=0, SignalSource=LCFA_profile 1
EventTableTriggerIO 10172: IOValue=[1], IRC5Controller=? -1, Operator=0, SignalSource=LCFA_profile 1
EventTableTriggerIO 10173: IOValue=[1], IRC5Controller=? -1, Operator=0, SignalSource=LCFA_profile 1
EventTableTriggerIO 10174: IOValue=[1], IRC5Controller=? -1, Operator=0, SignalSource=LCFA_profile 1
EventTableTriggerIO 10175: IOValue=[1], IRC5Controller=? -1, Operator=0, SignalSource=LCFA_profile 1
EventTableTriggerIO 10176: IOValue=[1], IRC5Controller=? -1, Operator=0, SignalSource=LCFA_profile 1
EventTableTriggerIO 10177: IOValue=[1], IRC5Controller=? -1, Operator=0, SignalSource=LCFA_profile 1
EventTableTriggerIO 10178: IOValue=[1], IRC5Controller=? -1, Operator=0, SignalSource=LCFA_profile 1
EventTableTriggerIO 10179: IOValue=[1], IRC5Controller=? -1, Operator=0, SignalSource=LCFA_profile 1
EventTableTriggerIO 10180: IOValue=[1], IRC5Controller=? -1, Operator=0, SignalSource=LCFA_profile 1
EventTableTriggerIO 10181: IOValue=[1], IRC5Controller=? -1, Operator=0, SignalSource=LCFA_profile 1
EventTableTriggerIO 10182: IOValue=[1], IRC5Controller=? -1, Operator=0, SignalSource=LCFA_profile 1
EventTableTriggerIO 10183: IOValue=[1], IRC5Controller=? -1, Operator=0, SignalSource=LCFA_profile 1
EventTableTriggerIO 10184: IOValue=[1], IRC5Controller=? -1, Operator=0, SignalSource=LCFA_profile 1
EventTableTriggerIO 10185: IOValue=[1], IRC5Controller=? -1, Operator=0, SignalSource=LCFA_profile 1
EventTableTriggerIO 10186: IOValue=[1], IRC5Controller=? -1, Operator=0, SignalSource=LCFA_profile 1
EventTableTriggerIO 10187: IOValue=[1], IRC5Controller=? -1, Operator=0, SignalSource=LCFA_profile 1
EventTableTriggerIO 10188: IOValue=[1], IRC5Controller=? -1, Operator=0, SignalSource=LCFA_profile 1
EventTableTriggerIO 10189: IOValue=[1], IRC5Controller=? -1, Operator=0, SignalSource=LCFA_profile 1
EventTableTriggerIO 10190: IOValue=[1], IRC5Controller=? -1, Operator=0, SignalSource=LCFA_profile 1
EventTableTriggerIO 10191: IOValue=[1], IRC5Controller=? -1, Operator=0, SignalSource=LCFA_profile 1
EventTableTriggerIO 10192: IOValue=[1], IRC5Controller=? -1, Operator=0, SignalSource=LCFA_profile 1
EventTableTriggerIO 10193: IOValue=[1], IRC5Controller=? -1, Operator=0, SignalSource=LCFA_profile 1
EventTableTriggerIO 10194: IOValue=[1], IRC5Controller=? -1, Operator=0, SignalSource=LCFA_profile 1
EventTableTriggerIO 10195: IOValue=[1], IRC5Controller=? -1, Operator=0, SignalSource=LCFA_profile 1
EventTableTriggerIO 10196: IOValue=[1], IRC5Controller=? -1, Operator=0, SignalSource=LCFA_profile 1
EventTableTriggerIO 10197: IOValue=[1], IRC5Controller=? -1, Operator=0, SignalSource=LCFA_profile 1
EventTableTriggerIO 10198: IOValue=[1], IRC5Controller=? -1, Operator=0, SignalSource=LCFA_profile 1
EventTableTriggerLogic 10199: layoutX=49, layoutY=26, Operand1=Pallet2.6 8213, Operand2=conv1_buffer_horizontal_open 8214, Operator=0, Delay=1000
EventTableTriggerLogic 10200: layoutX=49, layoutY=26, Operand1=Pallet2.6 8213, Operand2=conv1_buffer_horizontal_open 8214, Operator=0, Delay=1000
EventTableTriggerLogic 10201: layoutX=49, layoutY=26, Operand1=Pallet2.6 8213, Operand2=conv1_buffer_horizontal_open 8214, Operator=0, Delay=1000
EventTableTriggerLogic 10202: layoutX=49, layoutY=26, Operand1=Pallet2.6 8213, Operand2=conv1_buffer_horizontal_open 8214, Operator=0, Delay=1000
EventTableTriggerLogic 10203: layoutX=49, layoutY=26, Operand1=Pallet2.6 8213, Operand2=conv1_buffer_horizontal_open 8214, Operator=0, Delay=1000
EventTableTriggerLogic 10204: layoutX=49, layoutY=26, Operand1=Pallet2.6 8213, Operand2=conv1_buffer_horizontal_open 8214, Operator=0, Delay=1000
EventTableTriggerIO 10205: IOValue=[1], IRC5Controller=? -1, Operator=0, SignalSource=LCFA_profile 1
EventTableTriggerIO 10206: IOValue=[1], IRC5Controller=? -1, Operator=0, SignalSource=LCFA_profile 1
EventTableTriggerIO 10207: IOValue=[1], IRC5Controller=? -1, Operator=0, SignalSource=LCFA_profile 1
EventTableTriggerIO 10208: IOValue=[1], IRC5Controller=? -1, Operator=0, SignalSource=LCFA_profile 1
EventTableTriggerIO 10209: IOValue=[1], IRC5Controller=? -1, Operator=0, SignalSource=LCFA_profile 1
EventTableTriggerIO 10210: IOValue=[1], IRC5Controller=? -1, Operator=0, SignalSource=LCFA_profile 1
EventTableTriggerIO 10211: IOValue=[1], IRC5Controller=? -1, Operator=0, SignalSource=LCFA_profile 1
EventTableTriggerIO 10212: IOValue=[1], IRC5Controller=? -1, Operator=0, SignalSource=LCFA_profile 1
EventTableTriggerIO 10213: IOValue=[1], IRC5Controller=? -1, Operator=0, SignalSource=LCFA_profile 1
EventTableTriggerIO 10214: IOValue=[1], IRC5Controller=? -1, Operator=0, SignalSource=LCFA_profile 1
EventTableTriggerIO 10215: IOValue=[1], IRC5Controller=? -1, Operator=0, SignalSource=LCFA_profile 1
EventTableTriggerIO 10216: IOValue=[1], IRC5Controller=? -1, Operator=0, SignalSource=LCFA_profile 1
EventTableTriggerIO 10217: IOValue=[1], IRC5Controller=? -1, Operator=0, SignalSource=LCFA_profile 1
EventTableTriggerIO 10218: IOValue=[1], IRC5Controller=? -1, Operator=0, SignalSource=LCFA_profile 1
EventTableTriggerIO 10219: IOValue=[1], IRC5Controller=? -1, Operator=0, SignalSource=LCFA_profile 1
EventTableTriggerIO 10220: IOValue=[1], IRC5Controller=? -1, Operator=0, SignalSource=LCFA_profile 1
EventTableTriggerIO 10221: IOValue=[1], IRC5Controller=? -1, Operator=0, SignalSource=LCFA_profile 1
EventTableTriggerIO 10222: IOValue=[1], IRC5Controller=? -1, Operator=0, SignalSource=LCFA_profile 1
EventTableTriggerIO 10223: IOValue=[1], IRC5Controller=? -1, Operator=0, SignalSource=LCFA_profile 1
EventTableTriggerIO 10224: IOValue=[1], IRC5Controller=? -1, Operator=0, SignalSource=LCFA_profile 1
EventTableTriggerIO 10225: IOValue=[1], IRC5Controller=? -1, Operator=0, SignalSource=LCFA_profile 1
EventTableTriggerIO 10226: IOValue=[1], IRC5Controller=? -1, Operator=0, SignalSource=LCFA_profile 1
EventTableTriggerIO 10227: IOValue=[1], IRC5Controller=? -1, Operator=0, SignalSource=LCFA_profile 1
EventTableTriggerIO 10228: IOValue=[1], IRC5Controller=? -1, Operator=0, SignalSource=LCFA_profile 1
EventTableTriggerIO 10229: IOValue=[1], IRC5Controller=? -1, Operator=0, SignalSource=LCFA_profile 1
EventTableTriggerIO 10230: IOValue=[1], IRC5Controller=? -1, Operator=0, SignalSource=LCFA_profile 1
EventTableTriggerIO 10231: IOValue=[1], IRC5Controller=? -1, Operator=0, SignalSource=LCFA_profile 1
EventTableTriggerIO 10232: IOValue=[1], IRC5Controller=? -1, Operator=0, SignalSource=LCFA_profile 1
EventTableTriggerIO 10233: IOValue=[1], IRC5Controller=? -1, Operator=0, SignalSource=LCFA_profile 1
EventTableTriggerIO 10234: IOValue=[1], IRC5Controller=? -1, Operator=0, SignalSource=LCFA_profile 1
EventTableTriggerIO 10235: IOValue=[1], IRC5Controller=? -1, Operator=0, SignalSource=ALab_CellC_v1.0_4 5362
EventTableTriggerIO 10236: IOValue=[1], IRC5Controller=? -1, Operator=0, SignalSource=ALab_CellC_v1.0_4 5362
EventTableTriggerIO 10237: IOValue=[1], IRC5Controller=? -1, Operator=0, SignalSource=ALab_CellC_v1.0_4 5362
EventTableTriggerIO 10238: IOValue=[1], IRC5Controller=? -1, Operator=0, SignalSource=ALab_CellC_v1.0_4 5362
EventTableTriggerIO 10239: IOValue=[1], IRC5Controller=? -1, Operator=0, SignalSource=ALab_CellC_v1.0_4 5362
EventTableTriggerIO 10240: IOValue=[1], IRC5Controller=? -1, Operator=0, SignalSource=ALab_CellC_v1.0_4 5362
EventTableTriggerIO 10241: IOValue=[0], IRC5Controller=? -1, Operator=0, SignalSource=ALab_CellC_v1.0_4 5362
EventTableTriggerIO 10242: IOValue=[0], IRC5Controller=? -1, Operator=0, SignalSource=ALab_CellC_v1.0_4 5362
EventTableTriggerIO 10243: IOValue=[0], IRC5Controller=? -1, Operator=0, SignalSource=ALab_CellC_v1.0_4 5362
EventTableTriggerIO 10244: IOValue=[0], IRC5Controller=? -1, Operator=0, SignalSource=ALab_CellC_v1.0_4 5362
EventTableTriggerIO 10245: IOValue=[0], IRC5Controller=? -1, Operator=0, SignalSource=ALab_CellC_v1.0_4 5362
EventTableTriggerIO 10246: IOValue=[0], IRC5Controller=? -1, Operator=0, SignalSource=ALab_CellC_v1.0_4 5362
EventTableTriggerIO 10247: IOValue=[1], IRC5Controller=? -1, Operator=0, SignalSource=ALab_CellC_v1.0_4 5362
EventTableTriggerIO 10248: IOValue=[1], IRC5Controller=? -1, Operator=0, SignalSource=ALab_CellC_v1.0_4 5362
EventTableTriggerIO 10249: IOValue=[1], IRC5Controller=? -1, Operator=0, SignalSource=ALab_CellC_v1.0_4 5362
EventTableTriggerIO 10250: IOValue=[1], IRC5Controller=? -1, Operator=0, SignalSource=ALab_CellC_v1.0_4 5362
EventTableTriggerIO 10251: IOValue=[1], IRC5Controller=? -1, Operator=0, SignalSource=ALab_CellC_v1.0_4 5362
EventTableTriggerIO 10252: IOValue=[1], IRC5Controller=? -1, Operator=0, SignalSource=ALab_CellC_v1.0_4 5362
EventTableTriggerIO 10253: IOValue=[0], IRC5Controller=? -1, Operator=0, SignalSource=ALab_CellC_v1.0_4 5362
EventTableTriggerIO 10254: IOValue=[0], IRC5Controller=? -1, Operator=0, SignalSource=ALab_CellC_v1.0_4 5362
EventTableTriggerIO 10255: IOValue=[0], IRC5Controller=? -1, Operator=0, SignalSource=ALab_CellC_v1.0_4 5362
EventTableTriggerIO 10256: IOValue=[0], IRC5Controller=? -1, Operator=0, SignalSource=ALab_CellC_v1.0_4 5362
EventTableTriggerIO 10257: IOValue=[0], IRC5Controller=? -1, Operator=0, SignalSource=ALab_CellC_v1.0_4 5362
EventTableTriggerIO 10258: IOValue=[0], IRC5Controller=? -1, Operator=0, SignalSource=ALab_CellC_v1.0_4 5362
EventTableTriggerIO 10259: IOValue=[1], IRC5Controller=? -1, Operator=0, SignalSource=ALab_CellC_v1.0_4 5362
EventTableTriggerIO 10260: IOValue=[1], IRC5Controller=? -1, Operator=0, SignalSource=ALab_CellC_v1.0_4 5362
EventTableTriggerIO 10261: IOValue=[1], IRC5Controller=? -1, Operator=0, SignalSource=ALab_CellC_v1.0_4 5362
EventTableTriggerIO 10262: IOValue=[1], IRC5Controller=? -1, Operator=0, SignalSource=ALab_CellC_v1.0_4 5362
EventTableTriggerIO 10263: IOValue=[1], IRC5Controller=? -1, Operator=0, SignalSource=ALab_CellC_v1.0_4 5362
EventTableTriggerIO 10264: IOValue=[1], IRC5Controller=? -1, Operator=0, SignalSource=ALab_CellC_v1.0_4 5362
EventTableTriggerIO 10265: IOValue=[0], IRC5Controller=? -1, Operator=0, SignalSource=ALab_CellC_v1.0_4 5362
EventTableTriggerIO 10266: IOValue=[0], IRC5Controller=? -1, Operator=0, SignalSource=ALab_CellC_v1.0_4 5362
EventTableTriggerIO 10267: IOValue=[0], IRC5Controller=? -1, Operator=0, SignalSource=ALab_CellC_v1.0_4 5362
EventTableTriggerIO 10268: IOValue=[0], IRC5Controller=? -1, Operator=0, SignalSource=ALab_CellC_v1.0_4 5362
EventTableTriggerIO 10269: IOValue=[0], IRC5Controller=? -1, Operator=0, SignalSource=ALab_CellC_v1.0_4 5362
EventTableTriggerIO 10270: IOValue=[0], IRC5Controller=? -1, Operator=0, SignalSource=ALab_CellC_v1.0_4 5362
EventTableTriggerIO 10271: IOValue=[0], IRC5Controller=? -1, Operator=0, SignalSource=ALab_CellC_v1.0_4 5362
EventTableTriggerIO 10272: IOValue=[0], IRC5Controller=? -1, Operator=0, SignalSource=ALab_CellC_v1.0_4 5362
EventTableTriggerIO 10273: IOValue=[0], IRC5Controller=? -1, Operator=0, SignalSource=ALab_CellC_v1.0_4 5362
EventTableTriggerIO 10274: IOValue=[0], IRC5Controller=? -1, Operator=0, SignalSource=ALab_CellC_v1.0_4 5362
EventTableTriggerIO 10275: IOValue=[0], IRC5Controller=? -1, Operator=0, SignalSource=ALab_CellC_v1.0_4 5362
EventTableTriggerIO 10276: IOValue=[0], IRC5Controller=? -1, Operator=0, SignalSource=ALab_CellC_v1.0_4 5362
EventTableTriggerIO 10277: IOValue=[1], IRC5Controller=? -1, Operator=0, SignalSource=ALab_CellC_v1.0_4 5362
EventTableTriggerIO 10278: IOValue=[1], IRC5Controller=? -1, Operator=0, SignalSource=ALab_CellC_v1.0_4 5362
EventTableTriggerIO 10279: IOValue=[1], IRC5Controller=? -1, Operator=0, SignalSource=ALab_CellC_v1.0_4 5362
EventTableTriggerIO 10280: IOValue=[1], IRC5Controller=? -1, Operator=0, SignalSource=ALab_CellC_v1.0_4 5362
EventTableTriggerIO 10281: IOValue=[1], IRC5Controller=? -1, Operator=0, SignalSource=ALab_CellC_v1.0_4 5362
EventTableTriggerIO 10282: IOValue=[1], IRC5Controller=? -1, Operator=0, SignalSource=ALab_CellC_v1.0_4 5362
EventTableTriggerIO 10283: IOValue=[0], IRC5Controller=? -1, Operator=0, SignalSource=ALab_CellC_v1.0_4 5362
EventTableTriggerIO 10284: IOValue=[0], IRC5Controller=? -1, Operator=0, SignalSource=ALab_CellC_v1.0_4 5362
EventTableTriggerIO 10285: IOValue=[0], IRC5Controller=? -1, Operator=0, SignalSource=ALab_CellC_v1.0_4 5362
EventTableTriggerIO 10286: IOValue=[0], IRC5Controller=? -1, Operator=0, SignalSource=ALab_CellC_v1.0_4 5362
EventTableTriggerIO 10287: IOValue=[0], IRC5Controller=? -1, Operator=0, SignalSource=ALab_CellC_v1.0_4 5362
EventTableTriggerIO 10288: IOValue=[0], IRC5Controller=? -1, Operator=0, SignalSource=ALab_CellC_v1.0_4 5362
EventTableTriggerIO 10289: IOValue=[1], IRC5Controller=? -1, Operator=0, SignalSource=ALab_CellC_v1.0_4 5362
EventTableTriggerIO 10290: IOValue=[1], IRC5Controller=? -1, Operator=0, SignalSource=ALab_CellC_v1.0_4 5362
EventTableTriggerIO 10291: IOValue=[1], IRC5Controller=? -1, Operator=0, SignalSource=ALab_CellC_v1.0_4 5362
EventTableTriggerIO 10292: IOValue=[1], IRC5Controller=? -1, Operator=0, SignalSource=ALab_CellC_v1.0_4 5362
EventTableTriggerIO 10293: IOValue=[1], IRC5Controller=? -1, Operator=0, SignalSource=ALab_CellC_v1.0_4 5362
EventTableTriggerIO 10294: IOValue=[1], IRC5Controller=? -1, Operator=0, SignalSource=ALab_CellC_v1.0_4 5362
EventTableTriggerIO 10295: IOValue=[1], IRC5Controller=? -1, Operator=0, SignalSource=ALab_CellC_v1.0_4 5362
EventTableTriggerIO 10296: IOValue=[1], IRC5Controller=? -1, Operator=0, SignalSource=ALab_CellC_v1.0_4 5362
EventTableTriggerIO 10297: IOValue=[1], IRC5Controller=? -1, Operator=0, SignalSource=ALab_CellC_v1.0_4 5362
EventTableTriggerIO 10298: IOValue=[1], IRC5Controller=? -1, Operator=0, SignalSource=ALab_CellC_v1.0_4 5362
EventTableTriggerIO 10299: IOValue=[1], IRC5Controller=? -1, Operator=0, SignalSource=ALab_CellC_v1.0_4 5362
EventTableTriggerIO 10300: IOValue=[1], IRC5Controller=? -1, Operator=0, SignalSource=ALab_CellC_v1.0_4 5362
EventTableTriggerIO 10301: IOValue=[0], IRC5Controller=? -1, Operator=0, SignalSource=ALab_CellC_v1.0_4 5362
EventTableTriggerIO 10302: IOValue=[0], IRC5Controller=? -1, Operator=0, SignalSource=ALab_CellC_v1.0_4 5362
EventTableTriggerIO 10303: IOValue=[0], IRC5Controller=? -1, Operator=0, SignalSource=ALab_CellC_v1.0_4 5362
EventTableTriggerIO 10304: IOValue=[0], IRC5Controller=? -1, Operator=0, SignalSource=ALab_CellC_v1.0_4 5362
EventTableTriggerIO 10305: IOValue=[0], IRC5Controller=? -1, Operator=0, SignalSource=ALab_CellC_v1.0_4 5362
EventTableTriggerIO 10306: IOValue=[0], IRC5Controller=? -1, Operator=0, SignalSource=ALab_CellC_v1.0_4 5362
EventTableTriggerIO 10307: IOValue=[0], IRC5Controller=? -1, Operator=0, SignalSource=ALab_CellC_v1.0_4 5362
EventTableTriggerIO 10308: IOValue=[0], IRC5Controller=? -1, Operator=0, SignalSource=ALab_CellC_v1.0_4 5362
EventTableTriggerIO 10309: IOValue=[0], IRC5Controller=? -1, Operator=0, SignalSource=ALab_CellC_v1.0_4 5362
EventTableTriggerIO 10310: IOValue=[0], IRC5Controller=? -1, Operator=0, SignalSource=ALab_CellC_v1.0_4 5362
EventTableTriggerIO 10311: IOValue=[0], IRC5Controller=? -1, Operator=0, SignalSource=ALab_CellC_v1.0_4 5362
EventTableTriggerIO 10312: IOValue=[0], IRC5Controller=? -1, Operator=0, SignalSource=ALab_CellC_v1.0_4 5362
EventTableTriggerIO 10313: IOValue=[1], IRC5Controller=? -1, Operator=0, SignalSource=ALab_CellC_v1.0_4 5362
EventTableTriggerIO 10314: IOValue=[1], IRC5Controller=? -1, Operator=0, SignalSource=ALab_CellC_v1.0_4 5362
EventTableTriggerIO 10315: IOValue=[1], IRC5Controller=? -1, Operator=0, SignalSource=ALab_CellC_v1.0_4 5362
EventTableTriggerIO 10316: IOValue=[1], IRC5Controller=? -1, Operator=0, SignalSource=ALab_CellC_v1.0_4 5362
EventTableTriggerIO 10317: IOValue=[1], IRC5Controller=? -1, Operator=0, SignalSource=ALab_CellC_v1.0_4 5362
EventTableTriggerIO 10318: IOValue=[1], IRC5Controller=? -1, Operator=0, SignalSource=ALab_CellC_v1.0_4 5362
EventTableTriggerIO 10319: IOValue=[1], IRC5Controller=? -1, Operator=0, SignalSource=ALab_CellC_v1.0_4 5362
EventTableTriggerIO 10320: IOValue=[1], IRC5Controller=? -1, Operator=0, SignalSource=ALab_CellC_v1.0_4 5362
EventTableTriggerIO 10321: IOValue=[1], IRC5Controller=? -1, Operator=0, SignalSource=ALab_CellC_v1.0_4 5362
EventTableTriggerIO 10322: IOValue=[1], IRC5Controller=? -1, Operator=0, SignalSource=ALab_CellC_v1.0_4 5362
EventTableTriggerIO 10323: IOValue=[1], IRC5Controller=? -1, Operator=0, SignalSource=ALab_CellC_v1.0_4 5362
EventTableTriggerIO 10324: IOValue=[1], IRC5Controller=? -1, Operator=0, SignalSource=ALab_CellC_v1.0_4 5362
EventTableTriggerIO 10325: IOValue=[0], IRC5Controller=? -1, Operator=0, SignalSource=ALab_CellC_v1.0_4 5362
EventTableTriggerIO 10326: IOValue=[0], IRC5Controller=? -1, Operator=0, SignalSource=ALab_CellC_v1.0_4 5362
EventTableTriggerIO 10327: IOValue=[0], IRC5Controller=? -1, Operator=0, SignalSource=ALab_CellC_v1.0_4 5362
EventTableTriggerIO 10328: IOValue=[0], IRC5Controller=? -1, Operator=0, SignalSource=ALab_CellC_v1.0_4 5362
EventTableTriggerIO 10329: IOValue=[0], IRC5Controller=? -1, Operator=0, SignalSource=ALab_CellC_v1.0_4 5362
EventTableTriggerIO 10330: IOValue=[0], IRC5Controller=? -1, Operator=0, SignalSource=ALab_CellC_v1.0_4 5362
EventTableTriggerIO 10331: IOValue=[0], IRC5Controller=? -1, Operator=0, SignalSource=ALab_CellC_v1.0_4 5362
EventTableTriggerIO 10332: IOValue=[0], IRC5Controller=? -1, Operator=0, SignalSource=ALab_CellC_v1.0_4 5362
EventTableTriggerIO 10333: IOValue=[0], IRC5Controller=? -1, Operator=0, SignalSource=ALab_CellC_v1.0_4 5362
EventTableTriggerIO 10334: IOValue=[0], IRC5Controller=? -1, Operator=0, SignalSource=ALab_CellC_v1.0_4 5362
EventTableTriggerIO 10335: IOValue=[0], IRC5Controller=? -1, Operator=0, SignalSource=ALab_CellC_v1.0_4 5362
EventTableTriggerIO 10336: IOValue=[0], IRC5Controller=? -1, Operator=0, SignalSource=ALab_CellC_v1.0_4 5362
EventTableTriggerIO 10337: IOValue=[1], IRC5Controller=? -1, Operator=0, SignalSource=ALab_CellC_v1.0_4 5362
EventTableTriggerIO 10338: IOValue=[1], IRC5Controller=? -1, Operator=0, SignalSource=ALab_CellC_v1.0_4 5362
EventTableTriggerIO 10339: IOValue=[1], IRC5Controller=? -1, Operator=0, SignalSource=ALab_CellC_v1.0_4 5362
EventTableTriggerIO 10340: IOValue=[1], IRC5Controller=? -1, Operator=0, SignalSource=ALab_CellC_v1.0_4 5362
EventTableTriggerIO 10341: IOValue=[1], IRC5Controller=? -1, Operator=0, SignalSource=ALab_CellC_v1.0_4 5362
EventTableTriggerIO 10342: IOValue=[1], IRC5Controller=? -1, Operator=0, SignalSource=ALab_CellC_v1.0_4 5362
EventTableTriggerIO 10343: IOValue=[1], IRC5Controller=? -1, Operator=0, SignalSource=ALab_CellC_v1.0_4 5362
EventTableTriggerIO 10344: IOValue=[1], IRC5Controller=? -1, Operator=0, SignalSource=ALab_CellC_v1.0_4 5362
EventTableTriggerIO 10345: IOValue=[1], IRC5Controller=? -1, Operator=0, SignalSource=ALab_CellC_v1.0_4 5362
EventTableTriggerIO 10346: IOValue=[1], IRC5Controller=? -1, Operator=0, SignalSource=ALab_CellC_v1.0_4 5362
EventTableTriggerIO 10347: IOValue=[1], IRC5Controller=? -1, Operator=0, SignalSource=ALab_CellC_v1.0_4 5362
EventTableTriggerIO 10348: IOValue=[1], IRC5Controller=? -1, Operator=0, SignalSource=ALab_CellC_v1.0_4 5362
EventTableTriggerIO 10349: IOValue=[0], IRC5Controller=? -1, Operator=0, SignalSource=ALab_CellC_v1.0_4 5362
EventTableTriggerIO 10350: IOValue=[0], IRC5Controller=? -1, Operator=0, SignalSource=ALab_CellC_v1.0_4 5362
EventTableTriggerIO 10351: IOValue=[0], IRC5Controller=? -1, Operator=0, SignalSource=ALab_CellC_v1.0_4 5362
EventTableTriggerIO 10352: IOValue=[0], IRC5Controller=? -1, Operator=0, SignalSource=ALab_CellC_v1.0_4 5362
EventTableTriggerIO 10353: IOValue=[0], IRC5Controller=? -1, Operator=0, SignalSource=ALab_CellC_v1.0_4 5362
EventTableTriggerIO 10354: IOValue=[0], IRC5Controller=? -1, Operator=0, SignalSource=ALab_CellC_v1.0_4 5362
EventTableTriggerIO 10355: IOValue=[1], IRC5Controller=? -1, Operator=0, SignalSource=LCFA_profile 1
EventTableTriggerIO 10356: IOValue=[1], IRC5Controller=? -1, Operator=0, SignalSource=LCFA_profile 1
EventTableTriggerIO 10357: IOValue=[1], IRC5Controller=? -1, Operator=0, SignalSource=LCFA_profile 1
EventTableTriggerIO 10358: IOValue=[1], IRC5Controller=? -1, Operator=0, SignalSource=LCFA_profile 1
EventTableTriggerIO 10359: IOValue=[1], IRC5Controller=? -1, Operator=0, SignalSource=LCFA_profile 1
EventTableTriggerIO 10360: IOValue=[1], IRC5Controller=? -1, Operator=0, SignalSource=LCFA_profile 1
EventTableTriggerIO 10361: IOValue=[1], IRC5Controller=? -1, Operator=0, SignalSource=LCFA_profile 1
EventTableTriggerIO 10362: IOValue=[1], IRC5Controller=? -1, Operator=0, SignalSource=LCFA_profile 1
EventTableTriggerIO 10363: IOValue=[1], IRC5Controller=? -1, Operator=0, SignalSource=LCFA_profile 1
EventTableTriggerIO 10364: IOValue=[1], IRC5Controller=? -1, Operator=0, SignalSource=LCFA_profile 1
EventTableTriggerIO 10365: IOValue=[1], IRC5Controller=? -1, Operator=0, SignalSource=LCFA_profile 1
EventTableTriggerIO 10366: IOValue=[1], IRC5Controller=? -1, Operator=0, SignalSource=LCFA_profile 1
EventTableTriggerIO 10367: IOValue=[1], IRC5Controller=? -1, Operator=0, SignalSource=ALab_CellC_v1.0_4 5362
EventTableTriggerIO 10368: IOValue=[1], IRC5Controller=? -1, Operator=0, SignalSource=ALab_CellC_v1.0_4 5362
EventTableTriggerIO 10369: IOValue=[1], IRC5Controller=? -1, Operator=0, SignalSource=ALab_CellC_v1.0_4 5362
EventTableTriggerIO 10370: IOValue=[1], IRC5Controller=? -1, Operator=0, SignalSource=ALab_CellC_v1.0_4 5362
EventTableTriggerIO 10371: IOValue=[1], IRC5Controller=? -1, Operator=0, SignalSource=ALab_CellC_v1.0_4 5362
EventTableTriggerIO 10372: IOValue=[1], IRC5Controller=? -1, Operator=0, SignalSource=ALab_CellC_v1.0_4 5362
EventTableTriggerIO 10373: IOValue=[0], IRC5Controller=? -1, Operator=0, SignalSource=ALab_CellC_v1.0_4 5362
EventTableTriggerIO 10374: IOValue=[0], IRC5Controller=? -1, Operator=0, SignalSource=ALab_CellC_v1.0_4 5362
EventTableTriggerIO 10375: IOValue=[0], IRC5Controller=? -1, Operator=0, SignalSource=ALab_CellC_v1.0_4 5362
